KUKA KRL program: EPS_2_251349_CBMH081_A_20251001124256.src

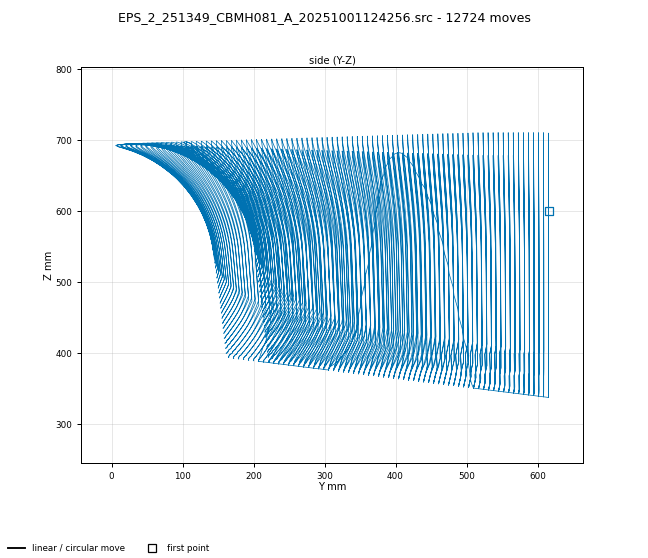
[picture p0: tool path of EPS_2_251349_CBMH081_A_20251001124256.src, 12724 of 12726 moves have a stored position in this frame; points joined in program order, loops and branches not executed]
&ACCESS RVP
&REL 4
&COMMENT QRS 19112012
&PARAM EDITMASK = *
DEF PART()
EXT BAS (BAS_COMMAND :IN,REAL :IN )
INT I
BAS (#INITMOV,0 )

;KUKA QRS Post kuka4.cps  Date:22-06-2017 !

File_ID=2858

QRS_PRE_INIT()

;Init var - Until changes are made in qrs_pre_init
Outlet_Square_prg=0
Inlet_1_Square_prg=0
Inlet_2_Square_prg=0
Inlet_3_Square_prg=0
Inlet_4_Square_prg=0
Inlet_5_Square_prg=0

Outlet_1={X 0.000, Y 517.920, Z 561.000, B 0.000, E1 0.000 }
Inlet_1={X 0.000, Y 520.260, Z 529.000, B 0.000, E1 170.000 }
Outlet_1_type=299
Inlet_1_type=299
;QRS#1=Sidecore dimensions
;QRS#2=300-12" PVC SDR 35
;QRS#3=300-12" PVC SDR 35
;QRS#4=
;QRS#5=
;QRS#6=
;QRS#7=
;QRS#8=
;QRS#9=16M PSX
;QRS#10=16M PSX
;QRS#11=
;QRS#12=
;QRS#13=
;QRS#14=
;QRS#15=
;QRS#16=1220x127x991 3,25'
;QRS#17=EPS Height
;QRS#18=710,5
;QRS#19=*
;QRS#20= UPDATED VERSION 22-06-2017
;QRS#21=*
Outlet_Square=0150
Inlet_1_Square=0150
Inlet_2_Square=0
Inlet_3_Square=0
Inlet_4_Square=0
Inlet_5_Square=0
Mill_Square=1
Outlet_Square_Prg=206
Inlet_1_Square_prg=206

QRS_INIT()

$ADVANCE=5

; T1
PTP {E1 173.61,E2 173.61}
PTP {X 0,Y 615.513,A -85,B 0,C 180,E1 173.61,E2 173.61,E3 0,E4 0,E5 0,E6 0}
QRS_SPEED_INIT()
LIN {X 0,Y 615.513,Z 600,A -85,B 0,C 180,E1 173.61,E2 173.61,E3 0,E4 0,E5 0,E6 0} C_VEL
LIN {X 0,Y 615.513,Z 347.498,A -85,B 0,C 180,E1 173.61,E2 173.61} C_VEL
LIN {X 0,Y 615.513,Z 339.324,A -85,B 0,C 180,E1 173.61,E2 173.61} C_VEL
LIN {X 0,Y 615.486,Z 337.324,A -85,B 0,C 180,E1 173.424,E2 173.424} C_VEL
LIN {X 0,Y 615.446,Z 337.318,A -85,B 0,C 180,E1 170.8,E2 170.8} C_VEL
LIN {X 0,Y 615.482,Z 337.311,A -85,B 0,C 180,E1 168.139,E2 168.139} C_VEL
LIN {X 0,Y 615.489,Z 337.325,A -85,B 0,C 180,E1 165.451,E2 165.451} C_VEL
LIN {X 0,Y 615.447,Z 337.317,A -85,B 0,C 180,E1 162.728,E2 162.728} C_VEL
LIN {X 0,Y 615.489,Z 337.312,A -85,B 0,C 180,E1 159.967,E2 159.967} C_VEL
LIN {X 0,Y 615.463,Z 337.321,A -85,B 0,C 180,E1 157.154,E2 157.154} C_VEL
LIN {X 0,Y 615.454,Z 337.32,A -85,B 0,C 180,E1 155.006,E2 155.006} C_VEL
LIN {X 0,Y 615.449,Z 337.318,A -85,B 0,C 180,E1 152.821,E2 152.821} C_VEL
LIN {X 0,Y 615.476,Z 337.311,A -85,B 0,C 180,E1 150.208,E2 150.208} C_VEL
LIN {X 0,Y 615.493,Z 337.324,A -85,B 0,C 180,E1 147.542,E2 147.542} C_VEL
LIN {X 0,Y 615.468,Z 337.322,A -85,B 0,C 180,E1 145.183,E2 145.183} C_VEL
LIN {X 0,Y 615.45,Z 337.317,A -85,B 0,C 180,E1 142.755,E2 142.755} C_VEL
LIN {X 0,Y 615.496,Z 337.311,A -85,B 0,C 180,E1 139.91,E2 139.91} C_VEL
LIN {X 0,Y 615.494,Z 337.319,A -85,B 0,C 180,E1 137.647,E2 137.647} C_VEL
LIN {X 0,Y 615.454,Z 337.319,A -85,B 0,C 180,E1 134.928,E2 134.928} C_VEL
LIN {X 0,Y 615.486,Z 337.31,A -85,B 0,C 180,E1 132.079,E2 132.079} C_VEL
LIN {X 0,Y 615.489,Z 337.317,A -85,B 0,C 180,E1 129.75,E2 129.75} C_VEL
LIN {X 0,Y 615.456,Z 337.319,A -85,B 0,C 180,E1 126.932,E2 126.932} C_VEL
LIN {X 0,Y 615.452,Z 337.316,A -85,B 0,C 180,E1 124.695,E2 124.695} C_VEL
LIN {X 0,Y 615.474,Z 337.453,A -85,B 0,C 180,E1 122.145,E2 122.145} C_VEL
LIN {X 0,Y 615.463,Z 358.452,A -85,B 0,C 180,E1 119.408,E2 119.408} C_VEL
LIN {X 0,Y 615.49,Z 368.008,A -85,B 0,C 180,E1 118.181,E2 118.181} C_VEL
LIN {X 0,Y 615.482,Z 532.764,A -85,B 0,C 180,E1 116.194,E2 116.194} C_VEL
LIN {X 0,Y 615.486,Z 547.148,A -85,B 0,C 180,E1 115.898,E2 115.898} C_VEL
LIN {X 0,Y 615.476,Z 562.128,A -85,B 0,C 180,E1 115.457,E2 115.457} C_VEL
LIN {X 0,Y 615.487,Z 576.373,A -85,B 0,C 180,E1 114.902,E2 114.902} C_VEL
LIN {X 0,Y 615.486,Z 590.475,A -85,B 0,C 180,E1 114.206,E2 114.206} C_VEL
LIN {X 0,Y 615.498,Z 602.734,A -85,B 0,C 180,E1 113.467,E2 113.467} C_VEL
LIN {X 0,Y 615.497,Z 614.806,A -85,B 0,C 180,E1 112.595,E2 112.595} C_VEL
LIN {X 0,Y 615.496,Z 626.273,A -85,B 0,C 180,E1 111.607,E2 111.607} C_VEL
LIN {X 0,Y 615.493,Z 636.516,A -85,B 0,C 180,E1 110.557,E2 110.557} C_VEL
LIN {X 0,Y 615.494,Z 646.441,A -85,B 0,C 180,E1 109.338,E2 109.338} C_VEL
LIN {X 0,Y 615.499,Z 653.657,A -85,B 0,C 180,E1 108.28,E2 108.28} C_VEL
LIN {X 0,Y 615.488,Z 661.243,A -85,B 0,C 180,E1 106.928,E2 106.928} C_VEL
LIN {X 0,Y 615.492,Z 667.287,A -85,B 0,C 180,E1 105.565,E2 105.565} C_VEL
LIN {X 0,Y 615.491,Z 670.83,A -85,B 0,C 180,E1 104.549,E2 104.549} C_VEL
LIN {X 0,Y 615.492,Z 674.376,A -85,B 0,C 180,E1 103.201,E2 103.201} C_VEL
LIN {X 0,Y 615.495,Z 676.661,A -85,B 0,C 180,E1 101.861,E2 101.861} C_VEL
LIN {X 0,Y 615.492,Z 677.759,A -85,B 0,C 180,E1 100.527,E2 100.527} C_VEL
LIN {X 0,Y 615.493,Z 677.697,A -85,B 0,C 180,E1 99.199,E2 99.199} C_VEL
LIN {X 0,Y 615.494,Z 676.457,A -85,B 0,C 180,E1 97.876,E2 97.876} C_VEL
LIN {X 0,Y 615.49,Z 674.047,A -85,B 0,C 180,E1 96.557,E2 96.557} C_VEL
LIN {X 0,Y 615.491,Z 670.446,A -85,B 0,C 180,E1 95.241,E2 95.241} C_VEL
LIN {X 0,Y 615.496,Z 665.591,A -85,B 0,C 180,E1 93.928,E2 93.928} C_VEL
LIN {X 0,Y 615.493,Z 659.363,A -85,B 0,C 180,E1 92.618,E2 92.618} C_VEL
LIN {X 0,Y 615.49,Z 651.592,A -85,B 0,C 180,E1 91.309,E2 91.309} C_VEL
LIN {X 0,Y 615.499,Z 643.35,A -85,B 0,C 180,E1 90.164,E2 90.164} C_VEL
LIN {X 0,Y 615.496,Z 633.468,A -85,B 0,C 180,E1 89.019,E2 89.019} C_VEL
LIN {X 0,Y 615.5,Z 623.429,A -85,B 0,C 180,E1 88.037,E2 88.037} C_VEL
LIN {X 0,Y 615.498,Z 611.464,A -85,B 0,C 180,E1 87.055,E2 87.055} C_VEL
LIN {X 0,Y 615.5,Z 599.577,A -85,B 0,C 180,E1 86.235,E2 86.235} C_VEL
LIN {X 0,Y 615.475,Z 586.657,A -85,B 0,C 180,E1 85.497,E2 85.497} C_VEL
LIN {X 0,Y 615.487,Z 572.479,A -85,B 0,C 180,E1 84.841,E2 84.841} C_VEL
LIN {X 0,Y 615.484,Z 557.682,A -85,B 0,C 180,E1 84.307,E2 84.307} C_VEL
LIN {X 0,Y 615.49,Z 543.934,A -85,B 0,C 180,E1 83.938,E2 83.938} C_VEL
LIN {X 0,Y 615.479,Z 529.603,A -85,B 0,C 180,E1 83.672,E2 83.672} C_VEL
LIN {X 0,Y 615.486,Z 367.825,A -85,B 0,C 180,E1 81.711,E2 81.711} C_VEL
LIN {X 0,Y 615.46,Z 346.644,A -85,B 0,C 180,E1 78.968,E2 78.968} C_VEL
LIN {X 0,Y 615.466,Z 337.313,A -85,B 0,C 180,E1 77.721,E2 77.721} C_VEL
LIN {X 0,Y 615.45,Z 337.315,A -85,B 0,C 180,E1 75.45,E2 75.45} C_VEL
LIN {X 0,Y 615.449,Z 337.316,A -85,B 0,C 180,E1 73.412,E2 73.412} C_VEL
LIN {X 0,Y 615.447,Z 337.316,A -85,B 0,C 180,E1 71.353,E2 71.353} C_VEL
LIN {X 0,Y 615.445,Z 337.317,A -85,B 0,C 180,E1 69.268,E2 69.268} C_VEL
LIN {X 0,Y 615.446,Z 337.318,A -85,B 0,C 180,E1 67.154,E2 67.154} C_VEL
LIN {X 0,Y 615.499,Z 337.324,A -85,B 0,C 180,E1 64.43,E2 64.43} C_VEL
LIN {X 0,Y 615.455,Z 337.314,A -85,B 0,C 180,E1 61.556,E2 61.556} C_VEL
LIN {X 0,Y 615.445,Z 337.32,A -85,B 0,C 180,E1 59.078,E2 59.078} C_VEL
LIN {X 0,Y 615.495,Z 337.326,A -85,B 0,C 180,E1 56.466,E2 56.466} C_VEL
LIN {X 0,Y 615.456,Z 337.314,A -85,B 0,C 180,E1 53.573,E2 53.573} C_VEL
LIN {X 0,Y 615.45,Z 337.321,A -85,B 0,C 180,E1 50.943,E2 50.943} C_VEL
LIN {X 0,Y 615.486,Z 337.325,A -85,B 0,C 180,E1 48.526,E2 48.526} C_VEL
LIN {X 0,Y 615.481,Z 337.312,A -85,B 0,C 180,E1 45.85,E2 45.85} C_VEL
LIN {X 0,Y 615.444,Z 337.317,A -85,B 0,C 180,E1 43.249,E2 43.249} C_VEL
LIN {X 0,Y 615.479,Z 337.324,A -85,B 0,C 180,E1 40.608,E2 40.608} C_VEL
LIN {X 0,Y 615.483,Z 337.315,A -85,B 0,C 180,E1 38.011,E2 38.011} C_VEL
LIN {X 0,Y 615.458,Z 337.314,A -85,B 0,C 180,E1 35.618,E2 35.618} C_VEL
LIN {X 0,Y 615.441,Z 337.318,A -85,B 0,C 180,E1 33.24,E2 33.24} C_VEL
LIN {X 0,Y 615.451,Z 337.321,A -85,B 0,C 180,E1 30.922,E2 30.922} C_VEL
LIN {X 0,Y 615.497,Z 337.325,A -85,B 0,C 180,E1 28.451,E2 28.451} C_VEL
LIN {X 0,Y 615.454,Z 337.315,A -85,B 0,C 180,E1 25.562,E2 25.562} C_VEL
LIN {X 0,Y 615.453,Z 337.315,A -85,B 0,C 180,E1 23.558,E2 23.558} C_VEL
LIN {X 0,Y 615.447,Z 337.316,A -85,B 0,C 180,E1 21.434,E2 21.434} C_VEL
LIN {X 0,Y 615.444,Z 337.317,A -85,B 0,C 180,E1 19.34,E2 19.34} C_VEL
LIN {X 0,Y 615.442,Z 337.317,A -85,B 0,C 180,E1 17.272,E2 17.272} C_VEL
LIN {X 0,Y 615.482,Z 337.324,A -85,B 0,C 180,E1 14.55,E2 14.55} C_VEL
LIN {X 0,Y 615.482,Z 337.312,A -85,B 0,C 180,E1 11.861,E2 11.861} C_VEL
LIN {X 0,Y 615.441,Z 337.318,A -85,B 0,C 180,E1 9.2,E2 9.2} C_VEL
LIN {X 0,Y 615.48,Z 337.324,A -85,B 0,C 180,E1 6.557,E2 6.557} C_VEL
LIN {X 0,Y 615.483,Z 337.314,A -85,B 0,C 180,E1 3.929,E2 3.929} C_VEL
LIN {X 0,Y 615.442,Z 337.317,A -85,B 0,C 180,E1 1.309,E2 1.309} C_VEL
LIN {X 0,Y 615.465,Z 337.323,A -85,B 0,C 180,E1 -1.308,E2 -1.308} C_VEL
LIN {X 0,Y 615.491,Z 337.316,A -85,B 0,C 180,E1 -3.928,E2 -3.928} C_VEL
LIN {X 0,Y 615.446,Z 337.316,A -85,B 0,C 180,E1 -6.557,E2 -6.557} C_VEL
LIN {X 0,Y 615.447,Z 337.316,A -85,B 0,C 180,E1 -8.537,E2 -8.537} C_VEL
LIN {X 0,Y 615.44,Z 337.319,A -85,B 0,C 180,E1 -10.864,E2 -10.864} C_VEL
LIN {X 0,Y 615.454,Z 337.322,A -85,B 0,C 180,E1 -13.202,E2 -13.202} C_VEL
LIN {X 0,Y 615.494,Z 337.316,A -85,B 0,C 180,E1 -15.905,E2 -15.905} C_VEL
LIN {X 0,Y 615.442,Z 337.317,A -85,B 0,C 180,E1 -18.647,E2 -18.647} C_VEL
LIN {X 0,Y 615.44,Z 337.318,A -85,B 0,C 180,E1 -20.732,E2 -20.732} C_VEL
LIN {X 0,Y 615.439,Z 337.319,A -85,B 0,C 180,E1 -22.846,E2 -22.846} C_VEL
LIN {X 0,Y 615.442,Z 337.32,A -85,B 0,C 180,E1 -24.994,E2 -24.994} C_VEL
LIN {X 0,Y 615.49,Z 337.317,A -85,B 0,C 180,E1 -27.915,E2 -27.915} C_VEL
LIN {X 0,Y 615.479,Z 337.313,A -85,B 0,C 180,E1 -30.16,E2 -30.16} C_VEL
LIN {X 0,Y 615.45,Z 337.316,A -85,B 0,C 180,E1 -32.459,E2 -32.459} C_VEL
LIN {X 0,Y 615.437,Z 337.319,A -85,B 0,C 180,E1 -34.818,E2 -34.818} C_VEL
LIN {X 0,Y 615.452,Z 337.323,A -85,B 0,C 180,E1 -37.245,E2 -37.245} C_VEL
LIN {X 0,Y 615.488,Z 337.313,A -85,B 0,C 180,E1 -40.089,E2 -40.089} C_VEL
LIN {X 0,Y 615.458,Z 337.315,A -85,B 0,C 180,E1 -42.355,E2 -42.355} C_VEL
LIN {X 0,Y 615.439,Z 337.32,A -85,B 0,C 180,E1 -44.927,E2 -44.927} C_VEL
LIN {X 0,Y 615.499,Z 337.325,A -85,B 0,C 180,E1 -47.648,E2 -47.648} C_VEL
LIN {X 0,Y 615.467,Z 337.315,A -85,B 0,C 180,E1 -50.248,E2 -50.248} C_VEL
LIN {X 0,Y 615.437,Z 337.318,A -85,B 0,C 180,E1 -52.754,E2 -52.754} C_VEL
LIN {X 0,Y 615.458,Z 337.322,A -85,B 0,C 180,E1 -55.303,E2 -55.303} C_VEL
LIN {X 0,Y 615.461,Z 337.315,A -85,B 0,C 180,E1 -58.313,E2 -58.313} C_VEL
LIN {X 0,Y 615.442,Z 337.317,A -85,B 0,C 180,E1 -60.591,E2 -60.591} C_VEL
LIN {X 0,Y 615.438,Z 337.32,A -85,B 0,C 180,E1 -62.964,E2 -62.964} C_VEL
LIN {X 0,Y 615.436,Z 337.373,A -85,B 0,C 180,E1 -64.846,E2 -64.846} C_VEL
LIN {X 0,Y 615.479,Z 359.775,A -85,B 0,C 180,E1 -67.404,E2 -67.404} C_VEL
LIN {X 0,Y 615.49,Z 384.221,A -85,B 0,C 180,E1 -70.141,E2 -70.141} C_VEL
LIN {X 0,Y 615.488,Z 399.033,A -85,B 0,C 180,E1 -71.762,E2 -71.762} C_VEL
LIN {X 0,Y 615.484,Z 565.218,A -85,B 0,C 180,E1 -73.769,E2 -73.769} C_VEL
LIN {X 0,Y 615.49,Z 580.71,A -85,B 0,C 180,E1 -74.095,E2 -74.095} C_VEL
LIN {X 0,Y 615.48,Z 596.048,A -85,B 0,C 180,E1 -74.562,E2 -74.562} C_VEL
LIN {X 0,Y 615.484,Z 609.752,A -85,B 0,C 180,E1 -75.113,E2 -75.113} C_VEL
LIN {X 0,Y 615.493,Z 624.045,A -85,B 0,C 180,E1 -75.833,E2 -75.833} C_VEL
LIN {X 0,Y 615.497,Z 636.897,A -85,B 0,C 180,E1 -76.631,E2 -76.631} C_VEL
LIN {X 0,Y 615.495,Z 649.254,A -85,B 0,C 180,E1 -77.554,E2 -77.554} C_VEL
LIN {X 0,Y 615.495,Z 659.606,A -85,B 0,C 180,E1 -78.473,E2 -78.473} C_VEL
LIN {X 0,Y 615.494,Z 669.183,A -85,B 0,C 180,E1 -79.473,E2 -79.473} C_VEL
LIN {X 0,Y 615.493,Z 678.577,A -85,B 0,C 180,E1 -80.636,E2 -80.636} C_VEL
LIN {X 0,Y 615.497,Z 686.38,A -85,B 0,C 180,E1 -81.794,E2 -81.794} C_VEL
LIN {X 0,Y 615.494,Z 693.609,A -85,B 0,C 180,E1 -83.102,E2 -83.102} C_VEL
LIN {X 0,Y 615.499,Z 699.436,A -85,B 0,C 180,E1 -84.43,E2 -84.43} C_VEL
LIN {X 0,Y 615.491,Z 702.86,A -85,B 0,C 180,E1 -85.415,E2 -85.415} C_VEL
LIN {X 0,Y 615.493,Z 706.318,A -85,B 0,C 180,E1 -86.727,E2 -86.727} C_VEL
LIN {X 0,Y 615.499,Z 708.593,A -85,B 0,C 180,E1 -88.037,E2 -88.037} C_VEL
LIN {X 0,Y 615.491,Z 709.741,A -85,B 0,C 180,E1 -89.346,E2 -89.346} C_VEL
LIN {X 0,Y 615.491,Z 709.741,A -85,B 0,C 180,E1 -90.654,E2 -90.654} C_VEL
LIN {X 0,Y 615.499,Z 708.593,A -85,B 0,C 180,E1 -91.963,E2 -91.963} C_VEL
LIN {X 0,Y 615.493,Z 706.318,A -85,B 0,C 180,E1 -93.273,E2 -93.273} C_VEL
LIN {X 0,Y 615.491,Z 702.86,A -85,B 0,C 180,E1 -94.584,E2 -94.584} C_VEL
LIN {X 0,Y 615.497,Z 698.142,A -85,B 0,C 180,E1 -95.898,E2 -95.898} C_VEL
LIN {X 0,Y 615.492,Z 692.03,A -85,B 0,C 180,E1 -97.216,E2 -97.216} C_VEL
LIN {X 0,Y 615.49,Z 684.333,A -85,B 0,C 180,E1 -98.537,E2 -98.537} C_VEL
LIN {X 0,Y 615.495,Z 676.114,A -85,B 0,C 180,E1 -99.696,E2 -99.696} C_VEL
LIN {X 0,Y 615.496,Z 665.898,A -85,B 0,C 180,E1 -100.892,E2 -100.892} C_VEL
LIN {X 0,Y 615.496,Z 656.067,A -85,B 0,C 180,E1 -101.861,E2 -101.861} C_VEL
LIN {X 0,Y 615.497,Z 643.947,A -85,B 0,C 180,E1 -102.865,E2 -102.865} C_VEL
LIN {X 0,Y 615.498,Z 631.797,A -85,B 0,C 180,E1 -103.706,E2 -103.706} C_VEL
LIN {X 0,Y 615.477,Z 618.379,A -85,B 0,C 180,E1 -104.473,E2 -104.473} C_VEL
LIN {X 0,Y 615.495,Z 603.847,A -85,B 0,C 180,E1 -105.141,E2 -105.141} C_VEL
LIN {X 0,Y 615.48,Z 589.615,A -85,B 0,C 180,E1 -105.65,E2 -105.65} C_VEL
LIN {X 0,Y 615.499,Z 575.154,A -85,B 0,C 180,E1 -106.035,E2 -106.035} C_VEL
LIN {X 0,Y 615.48,Z 560.677,A -85,B 0,C 180,E1 -106.296,E2 -106.296} C_VEL
LIN {X 0,Y 615.491,Z 398.712,A -85,B 0,C 180,E1 -108.258,E2 -108.258} C_VEL
LIN {X 0,Y 615.487,Z 373.248,A -85,B 0,C 180,E1 -111.081,E2 -111.081} C_VEL
LIN {X 0,Y 615.487,Z 349.309,A -85,B 0,C 180,E1 -113.783,E2 -113.783} C_VEL
LIN {X 0,Y 615.436,Z 337.319,A -85,B 0,C 180,E1 -115.171,E2 -115.171} C_VEL
LIN {X 0,Y 615.436,Z 337.319,A -85,B 0,C 180,E1 -117.18,E2 -117.18} C_VEL
LIN {X 0,Y 615.472,Z 337.314,A -85,B 0,C 180,E1 -119.792,E2 -119.792} C_VEL
LIN {X 0,Y 615.486,Z 337.324,A -85,B 0,C 180,E1 -122.458,E2 -122.458} C_VEL
LIN {X 0,Y 615.45,Z 337.322,A -85,B 0,C 180,E1 -124.818,E2 -124.818} C_VEL
LIN {X 0,Y 615.438,Z 337.318,A -85,B 0,C 180,E1 -127.246,E2 -127.246} C_VEL
LIN {X 0,Y 615.496,Z 337.316,A -85,B 0,C 180,E1 -130.09,E2 -130.09} C_VEL
LIN {X 0,Y 615.498,Z 337.325,A -85,B 0,C 180,E1 -132.352,E2 -132.352} C_VEL
LIN {X 0,Y 615.44,Z 337.319,A -85,B 0,C 180,E1 -135.073,E2 -135.073} C_VEL
LIN {X 0,Y 615.485,Z 337.313,A -85,B 0,C 180,E1 -137.92,E2 -137.92} C_VEL
LIN {X 0,Y 615.496,Z 337.321,A -85,B 0,C 180,E1 -140.251,E2 -140.251} C_VEL
LIN {X 0,Y 615.441,Z 337.319,A -85,B 0,C 180,E1 -143.069,E2 -143.069} C_VEL
LIN {X 0,Y 615.441,Z 337.317,A -85,B 0,C 180,E1 -145.306,E2 -145.306} C_VEL
LIN {X 0,Y 615.459,Z 337.315,A -85,B 0,C 180,E1 -147.674,E2 -147.674} C_VEL
LIN {X 0,Y 615.476,Z 337.323,A -85,B 0,C 180,E1 -150.593,E2 -150.593} C_VEL
LIN {X 0,Y 615.447,Z 337.32,A -85,B 0,C 180,E1 -152.963,E2 -152.963} C_VEL
LIN {X 0,Y 615.445,Z 337.32,A -85,B 0,C 180,E1 -155.007,E2 -155.007} C_VEL
LIN {X 0,Y 615.461,Z 337.314,A -85,B 0,C 180,E1 -157.661,E2 -157.661} C_VEL
LIN {X 0,Y 615.471,Z 337.323,A -85,B 0,C 180,E1 -160.662,E2 -160.662} C_VEL
LIN {X 0,Y 615.465,Z 337.322,A -85,B 0,C 180,E1 -162.729,E2 -162.729} C_VEL
LIN {X 0,Y 615.461,Z 337.322,A -85,B 0,C 180,E1 -164.774,E2 -164.774} C_VEL
LIN {X 0,Y 615.459,Z 337.322,A -85,B 0,C 180,E1 -166.798,E2 -166.798} C_VEL
LIN {X 0,Y 615.444,Z 337.319,A -85,B 0,C 180,E1 -169.134,E2 -169.134} C_VEL
LIN {X 0,Y 615.449,Z 337.315,A -85,B 0,C 180,E1 -171.463,E2 -171.463} C_VEL
LIN {X 0,Y 615.496,Z 337.314,A -85,B 0,C 180,E1 -174.102,E2 -174.102} C_VEL
LIN {X 0,Y 615.468,Z 337.322,A -85,B 0,C 180,E1 -176.727,E2 -176.727} C_VEL
LIN {X 0,Y 615.472,Z 337.323,A -85,B 0,C 180,E1 -178.692,E2 -178.692} C_VEL
LIN {X 0,Y 615.445,Z 337.317,A -85,B 0,C 180,E1 -181.309,E2 -181.309} C_VEL
LIN {X 0,Y 615.483,Z 337.312,A -85,B 0,C 180,E1 -183.929,E2 -183.929} C_VEL
LIN {X 0,Y 615.486,Z 337.324,A -85,B 0,C 180,E1 -186.576,E2 -186.576} C_VEL
LIN {X 0,Y 614.781,Z 337.464,A -85,B 0,C 180,E1 -187.122,E2 -187.122} C_VEL
LIN {X 0,Y 611.924,Z 337.883,A -85,B 0,C 180,E1 -188.007,E2 -188.007} C_VEL
LIN {X 0,Y 609.538,Z 338.19,A -85,B 0,C 180,E1 -188.72,E2 -188.72} C_VEL
LIN {X 0,Y 608.517,Z 338.305,A -85,B 0,C 180,E1 -189.27,E2 -189.27} C_VEL
LIN {X 0,Y 608.435,Z 338.314,A -85,B 0,C 180,E1 -189.456,E2 -189.456} C_VEL
LIN {X 0,Y 608.459,Z 338.314,A -85,B 0,C 180,E1 -192,E2 -192} C_VEL
LIN {X 0,Y 608.468,Z 338.317,A -85,B 0,C 180,E1 -194.721,E2 -194.721} C_VEL
LIN {X 0,Y 608.43,Z 338.315,A -85,B 0,C 180,E1 -197.478,E2 -197.478} C_VEL
LIN {X 0,Y 608.431,Z 338.314,A -85,B 0,C 180,E1 -199.572,E2 -199.572} C_VEL
LIN {X 0,Y 608.481,Z 338.318,A -85,B 0,C 180,E1 -202.405,E2 -202.405} C_VEL
LIN {X 0,Y 608.446,Z 338.322,A -85,B 0,C 180,E1 -204.572,E2 -204.572} C_VEL
LIN {X 0,Y 608.43,Z 338.316,A -85,B 0,C 180,E1 -207.198,E2 -207.198} C_VEL
LIN {X 0,Y 608.461,Z 338.312,A -85,B 0,C 180,E1 -209.78,E2 -209.78} C_VEL
LIN {X 0,Y 608.466,Z 338.322,A -85,B 0,C 180,E1 -212.523,E2 -212.523} C_VEL
LIN {X 0,Y 608.424,Z 338.316,A -85,B 0,C 180,E1 -215.279,E2 -215.279} C_VEL
LIN {X 0,Y 608.467,Z 338.316,A -85,B 0,C 180,E1 -218.24,E2 -218.24} C_VEL
LIN {X 0,Y 608.42,Z 338.317,A -85,B 0,C 180,E1 -221.18,E2 -221.18} C_VEL
LIN {X 0,Y 608.466,Z 338.312,A -85,B 0,C 180,E1 -223.87,E2 -223.87} C_VEL
LIN {X 0,Y 608.466,Z 338.319,A -85,B 0,C 180,E1 -226.692,E2 -226.692} C_VEL
LIN {X 0,Y 608.44,Z 338.32,A -85,B 0,C 180,E1 -228.822,E2 -228.822} C_VEL
LIN {X 0,Y 608.46,Z 338.312,A -85,B 0,C 180,E1 -231.761,E2 -231.761} C_VEL
LIN {X 0,Y 608.436,Z 338.322,A -85,B 0,C 180,E1 -234.722,E2 -234.722} C_VEL
LIN {X 0,Y 608.444,Z 338.316,A -85,B 0,C 180,E1 -237.12,E2 -237.12} C_VEL
LIN {X 0,Y 608.481,Z 338.475,A -85,B 0,C 180,E1 -237.722,E2 -237.722} C_VEL
LIN {X 0,Y 608.527,Z 357.408,A -85,B 0,C 180,E1 -240.224,E2 -240.224} C_VEL
LIN {X 0,Y 608.538,Z 367.98,A -85,B 0,C 180,E1 -241.603,E2 -241.603} C_VEL
LIN {X 0,Y 608.768,Z 378.048,A -85,B 0,C 180,E1 -241.732,E2 -241.732} C_VEL
LIN {X 0,Y 608.676,Z 533.346,A -85,B 0,C 180,E1 -243.629,E2 -243.629} C_VEL
LIN {X 0,Y 608.665,Z 549.358,A -85,B 0,C 180,E1 -243.975,E2 -243.975} C_VEL
LIN {X 0,Y 608.618,Z 563.717,A -85,B 0,C 180,E1 -244.416,E2 -244.416} C_VEL
LIN {X 0,Y 608.592,Z 577.624,A -85,B 0,C 180,E1 -244.979,E2 -244.979} C_VEL
LIN {X 0,Y 608.557,Z 591.482,A -85,B 0,C 180,E1 -245.682,E2 -245.682} C_VEL
LIN {X 0,Y 608.545,Z 604.931,A -85,B 0,C 180,E1 -246.52,E2 -246.52} C_VEL
LIN {X 0,Y 608.528,Z 617.115,A -85,B 0,C 180,E1 -247.436,E2 -247.436} C_VEL
LIN {X 0,Y 608.486,Z 628.833,A -85,B 0,C 180,E1 -248.487,E2 -248.487} C_VEL
LIN {X 0,Y 608.475,Z 639.142,A -85,B 0,C 180,E1 -249.594,E2 -249.594} C_VEL
LIN {X 0,Y 608.467,Z 648.398,A -85,B 0,C 180,E1 -250.781,E2 -250.781} C_VEL
LIN {X 0,Y 608.464,Z 656.297,A -85,B 0,C 180,E1 -252.003,E2 -252.003} C_VEL
LIN {X 0,Y 608.453,Z 662.751,A -85,B 0,C 180,E1 -253.216,E2 -253.216} C_VEL
LIN {X 0,Y 608.423,Z 668.603,A -85,B 0,C 180,E1 -254.593,E2 -254.593} C_VEL
LIN {X 0,Y 608.446,Z 673.082,A -85,B 0,C 180,E1 -255.994,E2 -255.994} C_VEL
LIN {X 0,Y 608.417,Z 676.06,A -85,B 0,C 180,E1 -257.322,E2 -257.322} C_VEL
LIN {X 0,Y 608.427,Z 677.88,A -85,B 0,C 180,E1 -258.675,E2 -258.675} C_VEL
LIN {X 0,Y 608.43,Z 678.499,A -85,B 0,C 180,E1 -260.022,E2 -260.022} C_VEL
LIN {X 0,Y 608.414,Z 677.916,A -85,B 0,C 180,E1 -261.363,E2 -261.363} C_VEL
LIN {X 0,Y 608.418,Z 676.173,A -85,B 0,C 180,E1 -262.7,E2 -262.7} C_VEL
LIN {X 0,Y 608.433,Z 673.251,A -85,B 0,C 180,E1 -264.033,E2 -264.033} C_VEL
LIN {X 0,Y 608.428,Z 669.105,A -85,B 0,C 180,E1 -265.362,E2 -265.362} C_VEL
LIN {X 0,Y 608.431,Z 663.65,A -85,B 0,C 180,E1 -266.689,E2 -266.689} C_VEL
LIN {X 0,Y 608.467,Z 656.739,A -85,B 0,C 180,E1 -268.014,E2 -268.014} C_VEL
LIN {X 0,Y 608.467,Z 648.185,A -85,B 0,C 180,E1 -269.338,E2 -269.338} C_VEL
LIN {X 0,Y 608.468,Z 639.143,A -85,B 0,C 180,E1 -270.496,E2 -270.496} C_VEL
LIN {X 0,Y 608.489,Z 628.289,A -85,B 0,C 180,E1 -271.655,E2 -271.655} C_VEL
LIN {X 0,Y 608.526,Z 617.195,A -85,B 0,C 180,E1 -272.648,E2 -272.648} C_VEL
LIN {X 0,Y 608.539,Z 605.104,A -85,B 0,C 180,E1 -273.559,E2 -273.559} C_VEL
LIN {X 0,Y 608.571,Z 591.843,A -85,B 0,C 180,E1 -274.388,E2 -274.388} C_VEL
LIN {X 0,Y 608.592,Z 578.944,A -85,B 0,C 180,E1 -275.052,E2 -275.052} C_VEL
LIN {X 0,Y 608.631,Z 564.807,A -85,B 0,C 180,E1 -275.633,E2 -275.633} C_VEL
LIN {X 0,Y 608.645,Z 549.57,A -85,B 0,C 180,E1 -276.11,E2 -276.11} C_VEL
LIN {X 0,Y 608.668,Z 534.404,A -85,B 0,C 180,E1 -276.441,E2 -276.441} C_VEL
LIN {X 0,Y 608.671,Z 500.168,A -85,B 0,C 180,E1 -276.88,E2 -276.88} C_VEL
LIN {X 0,Y 608.635,Z 368.605,A -85,B 0,C 180,E1 -278.477,E2 -278.477} C_VEL
LIN {X 0,Y 608.524,Z 367.812,A -85,B 0,C 180,E1 -278.51,E2 -278.51} C_VEL
LIN {X 0,Y 608.551,Z 347.627,A -85,B 0,C 180,E1 -281.152,E2 -281.152} C_VEL
LIN {X 0,Y 608.436,Z 338.316,A -85,B 0,C 180,E1 -282.402,E2 -282.402} C_VEL
LIN {X 0,Y 608.418,Z 338.317,A -85,B 0,C 180,E1 -284.722,E2 -284.722} C_VEL
LIN {X 0,Y 608.445,Z 338.323,A -85,B 0,C 180,E1 -287.477,E2 -287.477} C_VEL
LIN {X 0,Y 608.447,Z 338.313,A -85,B 0,C 180,E1 -290.275,E2 -290.275} C_VEL
LIN {X 0,Y 608.435,Z 338.314,A -85,B 0,C 180,E1 -292.469,E2 -292.469} C_VEL
LIN {X 0,Y 608.431,Z 338.315,A -85,B 0,C 180,E1 -294.572,E2 -294.572} C_VEL
LIN {X 0,Y 608.458,Z 338.316,A -85,B 0,C 180,E1 -297.202,E2 -297.202} C_VEL
LIN {X 0,Y 608.471,Z 338.313,A -85,B 0,C 180,E1 -299.971,E2 -299.971} C_VEL
LIN {X 0,Y 608.437,Z 338.315,A -85,B 0,C 180,E1 -302.881,E2 -302.881} C_VEL
LIN {X 0,Y 608.435,Z 338.32,A -85,B 0,C 180,E1 -305.278,E2 -305.278} C_VEL
LIN {X 0,Y 608.46,Z 338.312,A -85,B 0,C 180,E1 -308.239,E2 -308.239} C_VEL
LIN {X 0,Y 608.43,Z 338.319,A -85,B 0,C 180,E1 -311.179,E2 -311.179} C_VEL
LIN {X 0,Y 608.468,Z 338.315,A -85,B 0,C 180,E1 -313.87,E2 -313.87} C_VEL
LIN {X 0,Y 608.438,Z 338.314,A -85,B 0,C 180,E1 -316.695,E2 -316.695} C_VEL
LIN {X 0,Y 608.415,Z 338.317,A -85,B 0,C 180,E1 -318.82,E2 -318.82} C_VEL
LIN {X 0,Y 608.464,Z 338.318,A -85,B 0,C 180,E1 -321.76,E2 -321.76} C_VEL
LIN {X 0,Y 608.419,Z 338.316,A -85,B 0,C 180,E1 -324.72,E2 -324.72} C_VEL
LIN {X 0,Y 608.465,Z 338.32,A -85,B 0,C 180,E1 -327.478,E2 -327.478} C_VEL
LIN {X 0,Y 608.46,Z 338.312,A -85,B 0,C 180,E1 -330.22,E2 -330.22} C_VEL
LIN {X 0,Y 608.423,Z 338.316,A -85,B 0,C 180,E1 -332.803,E2 -332.803} C_VEL
LIN {X 0,Y 608.443,Z 338.321,A -85,B 0,C 180,E1 -335.428,E2 -335.428} C_VEL
LIN {X 0,Y 608.451,Z 338.313,A -85,B 0,C 180,E1 -338.307,E2 -338.307} C_VEL
LIN {X 0,Y 608.443,Z 338.317,A -85,B 0,C 180,E1 -341.13,E2 -341.13} C_VEL
LIN {X 0,Y 608.461,Z 338.316,A -85,B 0,C 180,E1 -343.906,E2 -343.906} C_VEL
LIN {X 0,Y 608.432,Z 338.315,A -85,B 0,C 180,E1 -346.643,E2 -346.643} C_VEL
LIN {X 0,Y 608.452,Z 338.318,A -85,B 0,C 180,E1 -349.35,E2 -349.35} C_VEL
LIN {X 0,Y 608.474,Z 338.313,A -85,B 0,C 180,E1 -352.033,E2 -352.033} C_VEL
LIN {X 0,Y 608.427,Z 338.315,A -85,B 0,C 180,E1 -354.697,E2 -354.697} C_VEL
LIN {X 0,Y 608.464,Z 338.317,A -85,B 0,C 180,E1 -357.352,E2 -357.352} C_VEL
LIN {X 0,Y 608.477,Z 338.313,A -85,B 0,C 180,E1 -360,E2 -360} C_VEL
LIN {X 0,Y 608.439,Z 338.313,A -85,B 0,C 180,E1 -362.648,E2 -362.648} C_VEL
LIN {X 0,Y 608.443,Z 338.319,A -85,B 0,C 180,E1 -365.302,E2 -365.302} C_VEL
LIN {X 0,Y 608.48,Z 338.313,A -85,B 0,C 180,E1 -367.967,E2 -367.967} C_VEL
LIN {X 0,Y 608.439,Z 338.315,A -85,B 0,C 180,E1 -370.939,E2 -370.939} C_VEL
LIN {X 0,Y 608.443,Z 338.319,A -85,B 0,C 180,E1 -373.357,E2 -373.357} C_VEL
LIN {X 0,Y 608.454,Z 338.315,A -85,B 0,C 180,E1 -376.094,E2 -376.094} C_VEL
LIN {X 0,Y 608.435,Z 338.315,A -85,B 0,C 180,E1 -378.87,E2 -378.87} C_VEL
LIN {X 0,Y 608.461,Z 338.321,A -85,B 0,C 180,E1 -381.692,E2 -381.692} C_VEL
LIN {X 0,Y 608.428,Z 338.315,A -85,B 0,C 180,E1 -384.572,E2 -384.572} C_VEL
LIN {X 0,Y 608.45,Z 338.316,A -85,B 0,C 180,E1 -387.202,E2 -387.202} C_VEL
LIN {X 0,Y 608.471,Z 338.315,A -85,B 0,C 180,E1 -389.972,E2 -389.972} C_VEL
LIN {X 0,Y 608.43,Z 338.315,A -85,B 0,C 180,E1 -392.881,E2 -392.881} C_VEL
LIN {X 0,Y 608.432,Z 338.319,A -85,B 0,C 180,E1 -395.278,E2 -395.278} C_VEL
LIN {X 0,Y 608.458,Z 338.313,A -85,B 0,C 180,E1 -398.239,E2 -398.239} C_VEL
LIN {X 0,Y 608.42,Z 338.319,A -85,B 0,C 180,E1 -401.179,E2 -401.179} C_VEL
LIN {X 0,Y 608.466,Z 338.317,A -85,B 0,C 180,E1 -403.87,E2 -403.87} C_VEL
LIN {X 0,Y 608.432,Z 338.315,A -85,B 0,C 180,E1 -406.695,E2 -406.695} C_VEL
LIN {X 0,Y 608.409,Z 338.318,A -85,B 0,C 180,E1 -408.819,E2 -408.819} C_VEL
LIN {X 0,Y 608.463,Z 338.32,A -85,B 0,C 180,E1 -411.76,E2 -411.76} C_VEL
LIN {X 0,Y 608.414,Z 338.317,A -85,B 0,C 180,E1 -414.72,E2 -414.72} C_VEL
LIN {X 0,Y 608.459,Z 338.319,A -85,B 0,C 180,E1 -417.478,E2 -417.478} C_VEL
LIN {X 0,Y 608.458,Z 338.314,A -85,B 0,C 180,E1 -420.22,E2 -420.22} C_VEL
LIN {X 0,Y 608.418,Z 338.317,A -85,B 0,C 180,E1 -422.804,E2 -422.804} C_VEL
LIN {X 0,Y 608.433,Z 338.45,A -85,B 0,C 180,E1 -424.662,E2 -424.662} C_VEL
LIN {X 0,Y 608.66,Z 349.305,A -85,B 0,C 180,E1 -425.933,E2 -425.933} C_VEL
LIN {X 0,Y 608.619,Z 373.247,A -85,B 0,C 180,E1 -428.67,E2 -428.67} C_VEL
LIN {X 0,Y 608.551,Z 398.721,A -85,B 0,C 180,E1 -431.526,E2 -431.526} C_VEL
LIN {X 0,Y 608.752,Z 404.044,A -85,B 0,C 180,E1 -431.614,E2 -431.614} C_VEL
LIN {X 0,Y 608.678,Z 565.217,A -85,B 0,C 180,E1 -433.582,E2 -433.582} C_VEL
LIN {X 0,Y 608.651,Z 580.709,A -85,B 0,C 180,E1 -433.911,E2 -433.911} C_VEL
LIN {X 0,Y 608.618,Z 596.047,A -85,B 0,C 180,E1 -434.383,E2 -434.383} C_VEL
LIN {X 0,Y 608.605,Z 609.754,A -85,B 0,C 180,E1 -434.94,E2 -434.94} C_VEL
LIN {X 0,Y 608.572,Z 623.235,A -85,B 0,C 180,E1 -435.624,E2 -435.624} C_VEL
LIN {X 0,Y 608.554,Z 635.663,A -85,B 0,C 180,E1 -436.39,E2 -436.39} C_VEL
LIN {X 0,Y 608.528,Z 648.282,A -85,B 0,C 180,E1 -437.324,E2 -437.324} C_VEL
LIN {X 0,Y 608.496,Z 659.747,A -85,B 0,C 180,E1 -438.339,E2 -438.339} C_VEL
LIN {X 0,Y 608.475,Z 669.387,A -85,B 0,C 180,E1 -439.35,E2 -439.35} C_VEL
LIN {X 0,Y 608.476,Z 678.853,A -85,B 0,C 180,E1 -440.527,E2 -440.527} C_VEL
LIN {X 0,Y 608.457,Z 686.729,A -85,B 0,C 180,E1 -441.698,E2 -441.698} C_VEL
LIN {X 0,Y 608.439,Z 694.087,A -85,B 0,C 180,E1 -443.034,E2 -443.034} C_VEL
LIN {X 0,Y 608.45,Z 699.923,A -85,B 0,C 180,E1 -444.366,E2 -444.366} C_VEL
LIN {X 0,Y 608.427,Z 703.383,A -85,B 0,C 180,E1 -445.362,E2 -445.362} C_VEL
LIN {X 0,Y 608.421,Z 706.885,A -85,B 0,C 180,E1 -446.689,E2 -446.689} C_VEL
LIN {X 0,Y 608.444,Z 709.191,A -85,B 0,C 180,E1 -448.014,E2 -448.014} C_VEL
LIN {X 0,Y 608.434,Z 710.351,A -85,B 0,C 180,E1 -449.338,E2 -449.338} C_VEL
LIN {X 0,Y 608.434,Z 710.351,A -85,B 0,C 180,E1 -450.662,E2 -450.662} C_VEL
LIN {X 0,Y 608.444,Z 709.191,A -85,B 0,C 180,E1 -451.986,E2 -451.986} C_VEL
LIN {X 0,Y 608.421,Z 706.885,A -85,B 0,C 180,E1 -453.311,E2 -453.311} C_VEL
LIN {X 0,Y 608.427,Z 703.383,A -85,B 0,C 180,E1 -454.638,E2 -454.638} C_VEL
LIN {X 0,Y 608.435,Z 698.608,A -85,B 0,C 180,E1 -455.967,E2 -455.967} C_VEL
LIN {X 0,Y 608.456,Z 692.426,A -85,B 0,C 180,E1 -457.299,E2 -457.299} C_VEL
LIN {X 0,Y 608.464,Z 684.654,A -85,B 0,C 180,E1 -458.636,E2 -458.636} C_VEL
LIN {X 0,Y 608.471,Z 676.37,A -85,B 0,C 180,E1 -459.809,E2 -459.809} C_VEL
LIN {X 0,Y 608.492,Z 665.652,A -85,B 0,C 180,E1 -461.063,E2 -461.063} C_VEL
LIN {X 0,Y 608.523,Z 654.274,A -85,B 0,C 180,E1 -462.168,E2 -462.168} C_VEL
LIN {X 0,Y 608.547,Z 642.854,A -85,B 0,C 180,E1 -463.1,E2 -463.1} C_VEL
LIN {X 0,Y 608.563,Z 630.446,A -85,B 0,C 180,E1 -463.95,E2 -463.95} C_VEL
LIN {X 0,Y 608.56,Z 616.858,A -85,B 0,C 180,E1 -464.718,E2 -464.718} C_VEL
LIN {X 0,Y 608.631,Z 602.79,A -85,B 0,C 180,E1 -465.359,E2 -465.359} C_VEL
LIN {X 0,Y 608.635,Z 588.3,A -85,B 0,C 180,E1 -465.874,E2 -465.874} C_VEL
LIN {X 0,Y 608.682,Z 573.042,A -85,B 0,C 180,E1 -466.269,E2 -466.269} C_VEL
LIN {X 0,Y 608.682,Z 557.166,A -85,B 0,C 180,E1 -466.533,E2 -466.533} C_VEL
LIN {X 0,Y 608.685,Z 399.645,A -85,B 0,C 180,E1 -468.442,E2 -468.442} C_VEL
LIN {X 0,Y 608.543,Z 398.536,A -85,B 0,C 180,E1 -468.495,E2 -468.495} C_VEL
LIN {X 0,Y 608.619,Z 373.248,A -85,B 0,C 180,E1 -471.33,E2 -471.33} C_VEL
LIN {X 0,Y 608.685,Z 347.17,A -85,B 0,C 180,E1 -474.313,E2 -474.313} C_VEL
LIN {X 0,Y 608.424,Z 338.318,A -85,B 0,C 180,E1 -475.356,E2 -475.356} C_VEL
LIN {X 0,Y 608.45,Z 338.323,A -85,B 0,C 180,E1 -478.267,E2 -478.267} C_VEL
LIN {X 0,Y 608.455,Z 338.319,A -85,B 0,C 180,E1 -480.546,E2 -480.546} C_VEL
LIN {X 0,Y 608.434,Z 338.317,A -85,B 0,C 180,E1 -482.881,E2 -482.881} C_VEL
LIN {X 0,Y 608.415,Z 338.317,A -85,B 0,C 180,E1 -485.28,E2 -485.28} C_VEL
LIN {X 0,Y 608.464,Z 338.319,A -85,B 0,C 180,E1 -488.24,E2 -488.24} C_VEL
LIN {X 0,Y 608.41,Z 338.318,A -85,B 0,C 180,E1 -491.18,E2 -491.18} C_VEL
LIN {X 0,Y 608.432,Z 338.315,A -85,B 0,C 180,E1 -493.305,E2 -493.305} C_VEL
LIN {X 0,Y 608.467,Z 338.317,A -85,B 0,C 180,E1 -496.131,E2 -496.131} C_VEL
LIN {X 0,Y 608.423,Z 338.319,A -85,B 0,C 180,E1 -498.821,E2 -498.821} C_VEL
LIN {X 0,Y 608.457,Z 338.313,A -85,B 0,C 180,E1 -501.761,E2 -501.761} C_VEL
LIN {X 0,Y 608.433,Z 338.32,A -85,B 0,C 180,E1 -504.722,E2 -504.722} C_VEL
LIN {X 0,Y 608.432,Z 338.315,A -85,B 0,C 180,E1 -507.119,E2 -507.119} C_VEL
LIN {X 0,Y 608.471,Z 338.314,A -85,B 0,C 180,E1 -510.028,E2 -510.028} C_VEL
LIN {X 0,Y 608.453,Z 338.316,A -85,B 0,C 180,E1 -512.798,E2 -512.798} C_VEL
LIN {X 0,Y 608.43,Z 338.315,A -85,B 0,C 180,E1 -515.428,E2 -515.428} C_VEL
LIN {X 0,Y 608.465,Z 338.32,A -85,B 0,C 180,E1 -518.309,E2 -518.309} C_VEL
LIN {X 0,Y 608.436,Z 338.315,A -85,B 0,C 180,E1 -521.13,E2 -521.13} C_VEL
LIN {X 0,Y 608.454,Z 338.314,A -85,B 0,C 180,E1 -523.906,E2 -523.906} C_VEL
LIN {X 0,Y 608.447,Z 338.32,A -85,B 0,C 180,E1 -526.643,E2 -526.643} C_VEL
LIN {X 0,Y 608.428,Z 338.315,A -85,B 0,C 180,E1 -529.35,E2 -529.35} C_VEL
LIN {X 0,Y 608.48,Z 338.312,A -85,B 0,C 180,E1 -532.033,E2 -532.033} C_VEL
LIN {X 0,Y 608.448,Z 338.319,A -85,B 0,C 180,E1 -534.698,E2 -534.698} C_VEL
LIN {X 0,Y 608.442,Z 338.313,A -85,B 0,C 180,E1 -537.352,E2 -537.352} C_VEL
LIN {X 0,Y 608.477,Z 338.312,A -85,B 0,C 180,E1 -540,E2 -540} C_VEL
LIN {X 0,Y 608.471,Z 338.317,A -85,B 0,C 180,E1 -542.648,E2 -542.648} C_VEL
LIN {X 0,Y 608.431,Z 338.315,A -85,B 0,C 180,E1 -545.302,E2 -545.302} C_VEL
LIN {X 0,Y 608.475,Z 338.312,A -85,B 0,C 180,E1 -547.967,E2 -547.967} C_VEL
LIN {X 0,Y 608.435,Z 338.314,A -85,B 0,C 180,E1 -549.456,E2 -549.456} C_VEL
LIN {X 0,Y 607.773,Z 338.401,A -85,B 0,C 180,E1 -550.008,E2 -550.008} C_VEL
LIN {X 0,Y 604.932,Z 338.754,A -85,B 0,C 180,E1 -550.905,E2 -550.905} C_VEL
LIN {X 0,Y 602.527,Z 339.055,A -85,B 0,C 180,E1 -551.627,E2 -551.627} C_VEL
LIN {X 0,Y 601.49,Z 339.185,A -85,B 0,C 180,E1 -552.183,E2 -552.183} C_VEL
LIN {X 0,Y 601.403,Z 339.194,A -85,B 0,C 180,E1 -552.372,E2 -552.372} C_VEL
LIN {X 0,Y 601.419,Z 339.192,A -85,B 0,C 180,E1 -554.898,E2 -554.898} C_VEL
LIN {X 0,Y 601.407,Z 339.193,A -85,B 0,C 180,E1 -556.987,E2 -556.987} C_VEL
LIN {X 0,Y 601.41,Z 339.19,A -85,B 0,C 180,E1 -559.1,E2 -559.1} C_VEL
LIN {X 0,Y 601.393,Z 339.192,A -85,B 0,C 180,E1 -561.24,E2 -561.24} C_VEL
LIN {X 0,Y 601.463,Z 339.187,A -85,B 0,C 180,E1 -564.141,E2 -564.141} C_VEL
LIN {X 0,Y 601.392,Z 339.193,A -85,B 0,C 180,E1 -567.114,E2 -567.114} C_VEL
LIN {X 0,Y 601.395,Z 339.191,A -85,B 0,C 180,E1 -569.395,E2 -569.395} C_VEL
LIN {X 0,Y 601.399,Z 339.191,A -85,B 0,C 180,E1 -571.728,E2 -571.728} C_VEL
LIN {X 0,Y 601.422,Z 339.192,A -85,B 0,C 180,E1 -574.119,E2 -574.119} C_VEL
LIN {X 0,Y 601.392,Z 339.202,A -85,B 0,C 180,E1 -576.584,E2 -576.584} C_VEL
LIN {X 0,Y 601.391,Z 339.193,A -85,B 0,C 180,E1 -579.129,E2 -579.129} C_VEL
LIN {X 0,Y 601.421,Z 339.189,A -85,B 0,C 180,E1 -581.766,E2 -581.766} C_VEL
LIN {X 0,Y 601.402,Z 339.202,A -85,B 0,C 180,E1 -584.533,E2 -584.533} C_VEL
LIN {X 0,Y 601.433,Z 339.195,A -85,B 0,C 180,E1 -586.428,E2 -586.428} C_VEL
LIN {X 0,Y 601.405,Z 339.192,A -85,B 0,C 180,E1 -589.125,E2 -589.125} C_VEL
LIN {X 0,Y 601.41,Z 339.19,A -85,B 0,C 180,E1 -591.731,E2 -591.731} C_VEL
LIN {X 0,Y 601.389,Z 339.198,A -85,B 0,C 180,E1 -594.245,E2 -594.245} C_VEL
LIN {X 0,Y 601.426,Z 339.198,A -85,B 0,C 180,E1 -596.686,E2 -596.686} C_VEL
LIN {X 0,Y 601.431,Z 339.31,A -85,B 0,C 180,E1 -597.559,E2 -597.559} C_VEL
LIN {X 0,Y 601.653,Z 344.666,A -85,B 0,C 180,E1 -598.288,E2 -598.288} C_VEL
LIN {X 0,Y 601.592,Z 364.647,A -85,B 0,C 180,E1 -600.943,E2 -600.943} C_VEL
LIN {X 0,Y 601.567,Z 367.973,A -85,B 0,C 180,E1 -601.38,E2 -601.38} C_VEL
LIN {X 0,Y 602.022,Z 371.233,A -85,B 0,C 180,E1 -601.436,E2 -601.436} C_VEL
LIN {X 0,Y 601.873,Z 532.501,A -85,B 0,C 180,E1 -603.425,E2 -603.425} C_VEL
LIN {X 0,Y 601.832,Z 548.146,A -85,B 0,C 180,E1 -603.755,E2 -603.755} C_VEL
LIN {X 0,Y 601.774,Z 563.452,A -85,B 0,C 180,E1 -604.225,E2 -604.225} C_VEL
LIN {X 0,Y 601.709,Z 577.829,A -85,B 0,C 180,E1 -604.812,E2 -604.812} C_VEL
LIN {X 0,Y 601.65,Z 591.769,A -85,B 0,C 180,E1 -605.529,E2 -605.529} C_VEL
LIN {X 0,Y 601.58,Z 605.73,A -85,B 0,C 180,E1 -606.414,E2 -606.414} C_VEL
LIN {X 0,Y 601.539,Z 618.113,A -85,B 0,C 180,E1 -607.368,E2 -607.368} C_VEL
LIN {X 0,Y 601.459,Z 629.376,A -85,B 0,C 180,E1 -608.403,E2 -608.403} C_VEL
LIN {X 0,Y 601.445,Z 639.217,A -85,B 0,C 180,E1 -609.479,E2 -609.479} C_VEL
LIN {X 0,Y 601.409,Z 648.777,A -85,B 0,C 180,E1 -610.724,E2 -610.724} C_VEL
LIN {X 0,Y 601.385,Z 656.609,A -85,B 0,C 180,E1 -611.96,E2 -611.96} C_VEL
LIN {X 0,Y 601.372,Z 662.163,A -85,B 0,C 180,E1 -613.012,E2 -613.012} C_VEL
LIN {X 0,Y 601.336,Z 668.156,A -85,B 0,C 180,E1 -614.407,E2 -614.407} C_VEL
LIN {X 0,Y 601.328,Z 672.676,A -85,B 0,C 180,E1 -615.792,E2 -615.792} C_VEL
LIN {X 0,Y 601.323,Z 675.862,A -85,B 0,C 180,E1 -617.17,E2 -617.17} C_VEL
LIN {X 0,Y 601.323,Z 677.778,A -85,B 0,C 180,E1 -618.54,E2 -618.54} C_VEL
LIN {X 0,Y 601.325,Z 678.473,A -85,B 0,C 180,E1 -619.903,E2 -619.903} C_VEL
LIN {X 0,Y 601.327,Z 677.999,A -85,B 0,C 180,E1 -621.261,E2 -621.261} C_VEL
LIN {X 0,Y 601.319,Z 676.368,A -85,B 0,C 180,E1 -622.613,E2 -622.613} C_VEL
LIN {X 0,Y 601.33,Z 673.563,A -85,B 0,C 180,E1 -623.962,E2 -623.962} C_VEL
LIN {X 0,Y 601.332,Z 669.539,A -85,B 0,C 180,E1 -625.307,E2 -625.307} C_VEL
LIN {X 0,Y 601.349,Z 664.205,A -85,B 0,C 180,E1 -626.65,E2 -626.65} C_VEL
LIN {X 0,Y 601.382,Z 657.417,A -85,B 0,C 180,E1 -627.991,E2 -627.991} C_VEL
LIN {X 0,Y 601.411,Z 649.029,A -85,B 0,C 180,E1 -629.33,E2 -629.33} C_VEL
LIN {X 0,Y 601.441,Z 640.123,A -85,B 0,C 180,E1 -630.502,E2 -630.502} C_VEL
LIN {X 0,Y 601.481,Z 629.5,A -85,B 0,C 180,E1 -631.674,E2 -631.674} C_VEL
LIN {X 0,Y 601.53,Z 617.622,A -85,B 0,C 180,E1 -632.762,E2 -632.762} C_VEL
LIN {X 0,Y 601.587,Z 605.612,A -85,B 0,C 180,E1 -633.684,E2 -633.684} C_VEL
LIN {X 0,Y 601.657,Z 592.459,A -85,B 0,C 180,E1 -634.522,E2 -634.522} C_VEL
LIN {X 0,Y 601.71,Z 577.844,A -85,B 0,C 180,E1 -635.278,E2 -635.278} C_VEL
LIN {X 0,Y 601.787,Z 563.441,A -85,B 0,C 180,E1 -635.865,E2 -635.865} C_VEL
LIN {X 0,Y 601.829,Z 547.557,A -85,B 0,C 180,E1 -636.35,E2 -636.35} C_VEL
LIN {X 0,Y 601.865,Z 532.706,A -85,B 0,C 180,E1 -636.662,E2 -636.662} C_VEL
LIN {X 0,Y 602.011,Z 370.318,A -85,B 0,C 180,E1 -638.666,E2 -638.666} C_VEL
LIN {X 0,Y 601.604,Z 367.772,A -85,B 0,C 180,E1 -638.735,E2 -638.735} C_VEL
LIN {X 0,Y 601.652,Z 347.265,A -85,B 0,C 180,E1 -641.454,E2 -641.454} C_VEL
LIN {X 0,Y 601.477,Z 339.648,A -85,B 0,C 180,E1 -642.484,E2 -642.484} C_VEL
LIN {X 0,Y 601.394,Z 339.196,A -85,B 0,C 180,E1 -642.571,E2 -642.571} C_VEL
LIN {X 0,Y 601.392,Z 339.194,A -85,B 0,C 180,E1 -644.898,E2 -644.898} C_VEL
LIN {X 0,Y 601.405,Z 339.193,A -85,B 0,C 180,E1 -646.987,E2 -646.987} C_VEL
LIN {X 0,Y 601.399,Z 339.197,A -85,B 0,C 180,E1 -649.81,E2 -649.81} C_VEL
LIN {X 0,Y 601.404,Z 339.19,A -85,B 0,C 180,E1 -652.683,E2 -652.683} C_VEL
LIN {X 0,Y 601.388,Z 339.194,A -85,B 0,C 180,E1 -654.879,E2 -654.879} C_VEL
LIN {X 0,Y 601.403,Z 339.198,A -85,B 0,C 180,E1 -657.359,E2 -657.359} C_VEL
LIN {X 0,Y 601.41,Z 339.191,A -85,B 0,C 180,E1 -660.165,E2 -660.165} C_VEL
LIN {X 0,Y 601.401,Z 339.19,A -85,B 0,C 180,E1 -662.711,E2 -662.711} C_VEL
LIN {X 0,Y 601.378,Z 339.197,A -85,B 0,C 180,E1 -665.109,E2 -665.109} C_VEL
LIN {X 0,Y 601.405,Z 339.198,A -85,B 0,C 180,E1 -667.421,E2 -667.421} C_VEL
LIN {X 0,Y 601.403,Z 339.193,A -85,B 0,C 180,E1 -669.996,E2 -669.996} C_VEL
LIN {X 0,Y 601.372,Z 339.194,A -85,B 0,C 180,E1 -672.674,E2 -672.674} C_VEL
LIN {X 0,Y 601.403,Z 339.2,A -85,B 0,C 180,E1 -675.479,E2 -675.479} C_VEL
LIN {X 0,Y 601.409,Z 339.19,A -85,B 0,C 180,E1 -678.409,E2 -678.409} C_VEL
LIN {X 0,Y 601.387,Z 339.193,A -85,B 0,C 180,E1 -680.871,E2 -680.871} C_VEL
LIN {X 0,Y 601.396,Z 339.199,A -85,B 0,C 180,E1 -683.741,E2 -683.741} C_VEL
LIN {X 0,Y 601.411,Z 339.189,A -85,B 0,C 180,E1 -686.685,E2 -686.685} C_VEL
LIN {X 0,Y 601.403,Z 339.193,A -85,B 0,C 180,E1 -689.057,E2 -689.057} C_VEL
LIN {X 0,Y 601.427,Z 339.194,A -85,B 0,C 180,E1 -691.372,E2 -691.372} C_VEL
LIN {X 0,Y 601.396,Z 339.19,A -85,B 0,C 180,E1 -694.38,E2 -694.38} C_VEL
LIN {X 0,Y 601.381,Z 339.192,A -85,B 0,C 180,E1 -696.588,E2 -696.588} C_VEL
LIN {X 0,Y 601.428,Z 339.196,A -85,B 0,C 180,E1 -699.478,E2 -699.478} C_VEL
LIN {X 0,Y 601.381,Z 339.193,A -85,B 0,C 180,E1 -702.311,E2 -702.311} C_VEL
LIN {X 0,Y 601.393,Z 339.192,A -85,B 0,C 180,E1 -704.408,E2 -704.408} C_VEL
LIN {X 0,Y 601.402,Z 339.194,A -85,B 0,C 180,E1 -707.171,E2 -707.171} C_VEL
LIN {X 0,Y 601.428,Z 339.192,A -85,B 0,C 180,E1 -709.905,E2 -709.905} C_VEL
LIN {X 0,Y 601.378,Z 339.193,A -85,B 0,C 180,E1 -712.614,E2 -712.614} C_VEL
LIN {X 0,Y 601.406,Z 339.195,A -85,B 0,C 180,E1 -715.308,E2 -715.308} C_VEL
LIN {X 0,Y 601.433,Z 339.191,A -85,B 0,C 180,E1 -717.991,E2 -717.991} C_VEL
LIN {X 0,Y 601.396,Z 339.191,A -85,B 0,C 180,E1 -720.669,E2 -720.669} C_VEL
LIN {X 0,Y 601.411,Z 339.195,A -85,B 0,C 180,E1 -723.349,E2 -723.349} C_VEL
LIN {X 0,Y 601.413,Z 339.192,A -85,B 0,C 180,E1 -726.037,E2 -726.037} C_VEL
LIN {X 0,Y 601.387,Z 339.192,A -85,B 0,C 180,E1 -728.738,E2 -728.738} C_VEL
LIN {X 0,Y 601.409,Z 339.198,A -85,B 0,C 180,E1 -731.458,E2 -731.458} C_VEL
LIN {X 0,Y 601.415,Z 339.19,A -85,B 0,C 180,E1 -734.205,E2 -734.205} C_VEL
LIN {X 0,Y 601.378,Z 339.195,A -85,B 0,C 180,E1 -736.987,E2 -736.987} C_VEL
LIN {X 0,Y 601.394,Z 339.199,A -85,B 0,C 180,E1 -739.81,E2 -739.81} C_VEL
LIN {X 0,Y 601.4,Z 339.19,A -85,B 0,C 180,E1 -742.683,E2 -742.683} C_VEL
LIN {X 0,Y 601.383,Z 339.193,A -85,B 0,C 180,E1 -744.879,E2 -744.879} C_VEL
LIN {X 0,Y 601.397,Z 339.197,A -85,B 0,C 180,E1 -747.358,E2 -747.358} C_VEL
LIN {X 0,Y 601.406,Z 339.192,A -85,B 0,C 180,E1 -750.165,E2 -750.165} C_VEL
LIN {X 0,Y 601.396,Z 339.191,A -85,B 0,C 180,E1 -752.711,E2 -752.711} C_VEL
LIN {X 0,Y 601.374,Z 339.196,A -85,B 0,C 180,E1 -755.109,E2 -755.109} C_VEL
LIN {X 0,Y 601.399,Z 339.198,A -85,B 0,C 180,E1 -757.422,E2 -757.422} C_VEL
LIN {X 0,Y 601.4,Z 339.195,A -85,B 0,C 180,E1 -759.996,E2 -759.996} C_VEL
LIN {X 0,Y 601.365,Z 339.195,A -85,B 0,C 180,E1 -762.674,E2 -762.674} C_VEL
LIN {X 0,Y 601.399,Z 339.199,A -85,B 0,C 180,E1 -765.479,E2 -765.479} C_VEL
LIN {X 0,Y 601.406,Z 339.191,A -85,B 0,C 180,E1 -768.409,E2 -768.409} C_VEL
LIN {X 0,Y 601.382,Z 339.194,A -85,B 0,C 180,E1 -770.871,E2 -770.871} C_VEL
LIN {X 0,Y 601.392,Z 339.201,A -85,B 0,C 180,E1 -773.741,E2 -773.741} C_VEL
LIN {X 0,Y 601.407,Z 339.19,A -85,B 0,C 180,E1 -776.685,E2 -776.685} C_VEL
LIN {X 0,Y 601.399,Z 339.193,A -85,B 0,C 180,E1 -779.057,E2 -779.057} C_VEL
LIN {X 0,Y 601.418,Z 339.195,A -85,B 0,C 180,E1 -781.372,E2 -781.372} C_VEL
LIN {X 0,Y 601.396,Z 339.195,A -85,B 0,C 180,E1 -784.427,E2 -784.427} C_VEL
LIN {X 0,Y 601.84,Z 343.461,A -85,B 0,C 180,E1 -784.956,E2 -784.956} C_VEL
LIN {X 0,Y 601.771,Z 365.894,A -85,B 0,C 180,E1 -787.568,E2 -787.568} C_VEL
LIN {X 0,Y 601.684,Z 390.492,A -85,B 0,C 180,E1 -790.378,E2 -790.378} C_VEL
LIN {X 0,Y 601.628,Z 398.844,A -85,B 0,C 180,E1 -791.32,E2 -791.32} C_VEL
LIN {X 0,Y 602.027,Z 403.039,A -85,B 0,C 180,E1 -791.389,E2 -791.389} C_VEL
LIN {X 0,Y 601.886,Z 564.282,A -85,B 0,C 180,E1 -793.377,E2 -793.377} C_VEL
LIN {X 0,Y 601.86,Z 579.884,A -85,B 0,C 180,E1 -793.704,E2 -793.704} C_VEL
LIN {X 0,Y 601.786,Z 594.789,A -85,B 0,C 180,E1 -794.158,E2 -794.158} C_VEL
LIN {X 0,Y 601.72,Z 609.757,A -85,B 0,C 180,E1 -794.764,E2 -794.764} C_VEL
LIN {X 0,Y 601.658,Z 623.231,A -85,B 0,C 180,E1 -795.455,E2 -795.455} C_VEL
LIN {X 0,Y 601.617,Z 636.448,A -85,B 0,C 180,E1 -796.283,E2 -796.283} C_VEL
LIN {X 0,Y 601.531,Z 648.283,A -85,B 0,C 180,E1 -797.174,E2 -797.174} C_VEL
LIN {X 0,Y 601.489,Z 659.747,A -85,B 0,C 180,E1 -798.201,E2 -798.201} C_VEL
LIN {X 0,Y 601.43,Z 669.388,A -85,B 0,C 180,E1 -799.224,E2 -799.224} C_VEL
LIN {X 0,Y 601.428,Z 678.854,A -85,B 0,C 180,E1 -800.414,E2 -800.414} C_VEL
LIN {X 0,Y 601.369,Z 686.73,A -85,B 0,C 180,E1 -801.6,E2 -801.6} C_VEL
LIN {X 0,Y 601.367,Z 694.087,A -85,B 0,C 180,E1 -802.951,E2 -802.951} C_VEL
LIN {X 0,Y 601.373,Z 699.924,A -85,B 0,C 180,E1 -804.299,E2 -804.299} C_VEL
LIN {X 0,Y 601.329,Z 703.383,A -85,B 0,C 180,E1 -805.307,E2 -805.307} C_VEL
LIN {X 0,Y 601.338,Z 706.886,A -85,B 0,C 180,E1 -806.65,E2 -806.65} C_VEL
LIN {X 0,Y 601.342,Z 709.192,A -85,B 0,C 180,E1 -807.991,E2 -807.991} C_VEL
LIN {X 0,Y 601.335,Z 710.35,A -85,B 0,C 180,E1 -809.33,E2 -809.33} C_VEL
LIN {X 0,Y 601.335,Z 710.35,A -85,B 0,C 180,E1 -810.67,E2 -810.67} C_VEL
LIN {X 0,Y 601.342,Z 709.192,A -85,B 0,C 180,E1 -812.009,E2 -812.009} C_VEL
LIN {X 0,Y 601.337,Z 706.886,A -85,B 0,C 180,E1 -813.35,E2 -813.35} C_VEL
LIN {X 0,Y 601.329,Z 703.383,A -85,B 0,C 180,E1 -814.693,E2 -814.693} C_VEL
LIN {X 0,Y 601.356,Z 698.608,A -85,B 0,C 180,E1 -816.038,E2 -816.038} C_VEL
LIN {X 0,Y 601.365,Z 692.425,A -85,B 0,C 180,E1 -817.386,E2 -817.386} C_VEL
LIN {X 0,Y 601.386,Z 684.653,A -85,B 0,C 180,E1 -818.738,E2 -818.738} C_VEL
LIN {X 0,Y 601.428,Z 676.37,A -85,B 0,C 180,E1 -819.925,E2 -819.925} C_VEL
LIN {X 0,Y 601.46,Z 665.932,A -85,B 0,C 180,E1 -821.165,E2 -821.165} C_VEL
LIN {X 0,Y 601.514,Z 656.192,A -85,B 0,C 180,E1 -822.14,E2 -822.14} C_VEL
LIN {X 0,Y 601.57,Z 644.015,A -85,B 0,C 180,E1 -823.168,E2 -823.168} C_VEL
LIN {X 0,Y 601.606,Z 632.077,A -85,B 0,C 180,E1 -824.012,E2 -824.012} C_VEL
LIN {X 0,Y 601.65,Z 618.526,A -85,B 0,C 180,E1 -824.805,E2 -824.805} C_VEL
LIN {X 0,Y 601.763,Z 603.842,A -85,B 0,C 180,E1 -825.495,E2 -825.495} C_VEL
LIN {X 0,Y 601.786,Z 589.617,A -85,B 0,C 180,E1 -826.016,E2 -826.016} C_VEL
LIN {X 0,Y 601.853,Z 574.718,A -85,B 0,C 180,E1 -826.419,E2 -826.419} C_VEL
LIN {X 0,Y 601.866,Z 559.746,A -85,B 0,C 180,E1 -826.689,E2 -826.689} C_VEL
LIN {X 0,Y 601.906,Z 400.45,A -85,B 0,C 180,E1 -828.647,E2 -828.647} C_VEL
LIN {X 0,Y 601.629,Z 398.715,A -85,B 0,C 180,E1 -828.695,E2 -828.695} C_VEL
LIN {X 0,Y 601.748,Z 373.248,A -85,B 0,C 180,E1 -831.586,E2 -831.586} C_VEL
LIN {X 0,Y 601.879,Z 349.049,A -85,B 0,C 180,E1 -834.386,E2 -834.386} C_VEL
LIN {X 0,Y 601.636,Z 340.326,A -85,B 0,C 180,E1 -835.423,E2 -835.423} C_VEL
LIN {X 0,Y 601.395,Z 339.197,A -85,B 0,C 180,E1 -835.573,E2 -835.573} C_VEL
LIN {X 0,Y 601.418,Z 339.195,A -85,B 0,C 180,E1 -838.628,E2 -838.628} C_VEL
LIN {X 0,Y 601.409,Z 339.19,A -85,B 0,C 180,E1 -841.453,E2 -841.453} C_VEL
LIN {X 0,Y 601.414,Z 339.196,A -85,B 0,C 180,E1 -844.119,E2 -844.119} C_VEL
LIN {X 0,Y 601.381,Z 339.2,A -85,B 0,C 180,E1 -846.585,E2 -846.585} C_VEL
LIN {X 0,Y 601.382,Z 339.193,A -85,B 0,C 180,E1 -849.129,E2 -849.129} C_VEL
LIN {X 0,Y 601.417,Z 339.19,A -85,B 0,C 180,E1 -851.766,E2 -851.766} C_VEL
LIN {X 0,Y 601.397,Z 339.199,A -85,B 0,C 180,E1 -854.533,E2 -854.533} C_VEL
LIN {X 0,Y 601.371,Z 339.194,A -85,B 0,C 180,E1 -857.414,E2 -857.414} C_VEL
LIN {X 0,Y 601.4,Z 339.195,A -85,B 0,C 180,E1 -860.004,E2 -860.004} C_VEL
LIN {X 0,Y 601.399,Z 339.197,A -85,B 0,C 180,E1 -862.623,E2 -862.623} C_VEL
LIN {X 0,Y 601.379,Z 339.194,A -85,B 0,C 180,E1 -865.066,E2 -865.066} C_VEL
LIN {X 0,Y 601.404,Z 339.19,A -85,B 0,C 180,E1 -867.483,E2 -867.483} C_VEL
LIN {X 0,Y 601.408,Z 339.191,A -85,B 0,C 180,E1 -869.855,E2 -869.855} C_VEL
LIN {X 0,Y 601.399,Z 339.197,A -85,B 0,C 180,E1 -872.641,E2 -872.641} C_VEL
LIN {X 0,Y 601.385,Z 339.193,A -85,B 0,C 180,E1 -875.121,E2 -875.121} C_VEL
LIN {X 0,Y 601.397,Z 339.195,A -85,B 0,C 180,E1 -878.04,E2 -878.04} C_VEL
LIN {X 0,Y 601.407,Z 339.193,A -85,B 0,C 180,E1 -880.901,E2 -880.901} C_VEL
LIN {X 0,Y 601.413,Z 339.19,A -85,B 0,C 180,E1 -883.713,E2 -883.713} C_VEL
LIN {X 0,Y 601.407,Z 339.2,A -85,B 0,C 180,E1 -886.484,E2 -886.484} C_VEL
LIN {X 0,Y 601.387,Z 339.193,A -85,B 0,C 180,E1 -889.224,E2 -889.224} C_VEL
LIN {X 0,Y 601.439,Z 339.188,A -85,B 0,C 180,E1 -891.939,E2 -891.939} C_VEL
LIN {X 0,Y 601.415,Z 339.196,A -85,B 0,C 180,E1 -894.636,E2 -894.636} C_VEL
LIN {X 0,Y 601.412,Z 339.189,A -85,B 0,C 180,E1 -897.321,E2 -897.321} C_VEL
LIN {X 0,Y 601.445,Z 339.188,A -85,B 0,C 180,E1 -900,E2 -900} C_VEL
LIN {X 0,Y 601.434,Z 339.193,A -85,B 0,C 180,E1 -902.679,E2 -902.679} C_VEL
LIN {X 0,Y 601.399,Z 339.191,A -85,B 0,C 180,E1 -905.365,E2 -905.365} C_VEL
LIN {X 0,Y 601.438,Z 339.189,A -85,B 0,C 180,E1 -908.061,E2 -908.061} C_VEL
LIN {X 0,Y 601.401,Z 339.193,A -85,B 0,C 180,E1 -910.999,E2 -910.999} C_VEL
LIN {X 0,Y 601.403,Z 339.194,A -85,B 0,C 180,E1 -912.372,E2 -912.372} C_VEL
LIN {X 0,Y 600.732,Z 339.278,A -85,B 0,C 180,E1 -912.931,E2 -912.931} C_VEL
LIN {X 0,Y 597.881,Z 339.632,A -85,B 0,C 180,E1 -913.839,E2 -913.839} C_VEL
LIN {X 0,Y 595.473,Z 339.938,A -85,B 0,C 180,E1 -914.569,E2 -914.569} C_VEL
LIN {X 0,Y 594.436,Z 340.06,A -85,B 0,C 180,E1 -915.133,E2 -915.133} C_VEL
LIN {X 0,Y 594.349,Z 340.069,A -85,B 0,C 180,E1 -915.324,E2 -915.324} C_VEL
LIN {X 0,Y 594.373,Z 340.067,A -85,B 0,C 180,E1 -917.194,E2 -917.194} C_VEL
LIN {X 0,Y 594.37,Z 340.068,A -85,B 0,C 180,E1 -920.054,E2 -920.054} C_VEL
LIN {X 0,Y 594.355,Z 340.071,A -85,B 0,C 180,E1 -922.968,E2 -922.968} C_VEL
LIN {X 0,Y 594.354,Z 340.068,A -85,B 0,C 180,E1 -925.194,E2 -925.194} C_VEL
LIN {X 0,Y 594.374,Z 340.072,A -85,B 0,C 180,E1 -928.228,E2 -928.228} C_VEL
LIN {X 0,Y 594.379,Z 340.074,A -85,B 0,C 180,E1 -930.56,E2 -930.56} C_VEL
LIN {X 0,Y 594.379,Z 340.069,A -85,B 0,C 180,E1 -932.951,E2 -932.951} C_VEL
LIN {X 0,Y 594.328,Z 340.071,A -85,B 0,C 180,E1 -935.411,E2 -935.411} C_VEL
LIN {X 0,Y 594.375,Z 340.068,A -85,B 0,C 180,E1 -937.942,E2 -937.942} C_VEL
LIN {X 0,Y 594.367,Z 340.073,A -85,B 0,C 180,E1 -940.821,E2 -940.821} C_VEL
LIN {X 0,Y 594.353,Z 340.069,A -85,B 0,C 180,E1 -943.301,E2 -943.301} C_VEL
LIN {X 0,Y 594.364,Z 340.071,A -85,B 0,C 180,E1 -946.162,E2 -946.162} C_VEL
LIN {X 0,Y 594.381,Z 340.076,A -85,B 0,C 180,E1 -948.536,E2 -948.536} C_VEL
LIN {X 0,Y 594.37,Z 340.068,A -85,B 0,C 180,E1 -951.298,E2 -951.298} C_VEL
LIN {X 0,Y 594.35,Z 340.07,A -85,B 0,C 180,E1 -953.755,E2 -953.755} C_VEL
LIN {X 0,Y 594.381,Z 340.072,A -85,B 0,C 180,E1 -956.239,E2 -956.239} C_VEL
LIN {X 0,Y 594.408,Z 340.232,A -85,B 0,C 180,E1 -957.404,E2 -957.404} C_VEL
LIN {X 0,Y 594.77,Z 343.595,A -85,B 0,C 180,E1 -957.877,E2 -957.877} C_VEL
LIN {X 0,Y 594.641,Z 364.027,A -85,B 0,C 180,E1 -960.628,E2 -960.628} C_VEL
LIN {X 0,Y 594.648,Z 367.911,A -85,B 0,C 180,E1 -961.147,E2 -961.147} C_VEL
LIN {X 0,Y 595.307,Z 372.232,A -85,B 0,C 180,E1 -961.231,E2 -961.231} C_VEL
LIN {X 0,Y 595.068,Z 533.108,A -85,B 0,C 180,E1 -963.239,E2 -963.239} C_VEL
LIN {X 0,Y 595.02,Z 548.72,A -85,B 0,C 180,E1 -963.578,E2 -963.578} C_VEL
LIN {X 0,Y 594.94,Z 563.093,A -85,B 0,C 180,E1 -964.026,E2 -964.026} C_VEL
LIN {X 0,Y 594.838,Z 578.037,A -85,B 0,C 180,E1 -964.641,E2 -964.641} C_VEL
LIN {X 0,Y 594.734,Z 592.57,A -85,B 0,C 180,E1 -965.402,E2 -965.402} C_VEL
LIN {X 0,Y 594.637,Z 605.184,A -85,B 0,C 180,E1 -966.214,E2 -966.214} C_VEL
LIN {X 0,Y 594.553,Z 618.195,A -85,B 0,C 180,E1 -967.223,E2 -967.223} C_VEL
LIN {X 0,Y 594.443,Z 629.89,A -85,B 0,C 180,E1 -968.317,E2 -968.317} C_VEL
LIN {X 0,Y 594.394,Z 639.666,A -85,B 0,C 180,E1 -969.405,E2 -969.405} C_VEL
LIN {X 0,Y 594.346,Z 649.14,A -85,B 0,C 180,E1 -970.665,E2 -970.665} C_VEL
LIN {X 0,Y 594.304,Z 656.919,A -85,B 0,C 180,E1 -971.915,E2 -971.915} C_VEL
LIN {X 0,Y 594.274,Z 664.026,A -85,B 0,C 180,E1 -973.322,E2 -973.322} C_VEL
LIN {X 0,Y 594.261,Z 668.987,A -85,B 0,C 180,E1 -974.568,E2 -974.568} C_VEL
LIN {X 0,Y 594.265,Z 673.028,A -85,B 0,C 180,E1 -975.876,E2 -975.876} C_VEL
LIN {X 0,Y 594.242,Z 675.644,A -85,B 0,C 180,E1 -977.014,E2 -977.014} C_VEL
LIN {X 0,Y 594.234,Z 677.641,A -85,B 0,C 180,E1 -978.401,E2 -978.401} C_VEL
LIN {X 0,Y 594.227,Z 678.446,A -85,B 0,C 180,E1 -979.781,E2 -979.781} C_VEL
LIN {X 0,Y 594.223,Z 678.082,A -85,B 0,C 180,E1 -981.155,E2 -981.155} C_VEL
LIN {X 0,Y 594.223,Z 676.563,A -85,B 0,C 180,E1 -982.525,E2 -982.525} C_VEL
LIN {X 0,Y 594.235,Z 673.875,A -85,B 0,C 180,E1 -983.89,E2 -983.89} C_VEL
LIN {X 0,Y 594.236,Z 669.956,A -85,B 0,C 180,E1 -985.251,E2 -985.251} C_VEL
LIN {X 0,Y 594.271,Z 664.707,A -85,B 0,C 180,E1 -986.61,E2 -986.61} C_VEL
LIN {X 0,Y 594.296,Z 658.051,A -85,B 0,C 180,E1 -987.967,E2 -987.967} C_VEL
LIN {X 0,Y 594.333,Z 650.921,A -85,B 0,C 180,E1 -989.153,E2 -989.153} C_VEL
LIN {X 0,Y 594.387,Z 642.406,A -85,B 0,C 180,E1 -990.339,E2 -990.339} C_VEL
LIN {X 0,Y 594.459,Z 632.223,A -85,B 0,C 180,E1 -991.524,E2 -991.524} C_VEL
LIN {X 0,Y 594.528,Z 621.861,A -85,B 0,C 180,E1 -992.541,E2 -992.541} C_VEL
LIN {X 0,Y 594.602,Z 609.52,A -85,B 0,C 180,E1 -993.558,E2 -993.558} C_VEL
LIN {X 0,Y 594.726,Z 597.173,A -85,B 0,C 180,E1 -994.405,E2 -994.405} C_VEL
LIN {X 0,Y 594.788,Z 583.728,A -85,B 0,C 180,E1 -995.169,E2 -995.169} C_VEL
LIN {X 0,Y 594.906,Z 569.814,A -85,B 0,C 180,E1 -995.806,E2 -995.806} C_VEL
LIN {X 0,Y 595.002,Z 555.237,A -85,B 0,C 180,E1 -996.324,E2 -996.324} C_VEL
LIN {X 0,Y 595.062,Z 540.778,A -85,B 0,C 180,E1 -996.703,E2 -996.703} C_VEL
LIN {X 0,Y 595.105,Z 525.088,A -85,B 0,C 180,E1 -996.967,E2 -996.967} C_VEL
LIN {X 0,Y 595.219,Z 370.867,A -85,B 0,C 180,E1 -998.879,E2 -998.879} C_VEL
LIN {X 0,Y 594.643,Z 367.898,A -85,B 0,C 180,E1 -998.945,E2 -998.945} C_VEL
LIN {X 0,Y 594.753,Z 346.921,A -85,B 0,C 180,E1 -1001.762,E2 -1001.762} C_VEL
LIN {X 0,Y 594.68,Z 341.839,A -85,B 0,C 180,E1 -1002.456,E2 -1002.456} C_VEL
LIN {X 0,Y 594.343,Z 340.076,A -85,B 0,C 180,E1 -1002.723,E2 -1002.723} C_VEL
LIN {X 0,Y 594.348,Z 340.074,A -85,B 0,C 180,E1 -1005.079,E2 -1005.079} C_VEL
LIN {X 0,Y 594.374,Z 340.072,A -85,B 0,C 180,E1 -1007.194,E2 -1007.194} C_VEL
LIN {X 0,Y 594.365,Z 340.07,A -85,B 0,C 180,E1 -1010.054,E2 -1010.054} C_VEL
LIN {X 0,Y 594.354,Z 340.071,A -85,B 0,C 180,E1 -1012.968,E2 -1012.968} C_VEL
LIN {X 0,Y 594.371,Z 340.071,A -85,B 0,C 180,E1 -1015.193,E2 -1015.193} C_VEL
LIN {X 0,Y 594.351,Z 340.08,A -85,B 0,C 180,E1 -1017.519,E2 -1017.519} C_VEL
LIN {X 0,Y 594.373,Z 340.067,A -85,B 0,C 180,E1 -1020.325,E2 -1020.325} C_VEL
LIN {X 0,Y 594.378,Z 340.067,A -85,B 0,C 180,E1 -1022.95,E2 -1022.95} C_VEL
LIN {X 0,Y 594.329,Z 340.08,A -85,B 0,C 180,E1 -1025.411,E2 -1025.411} C_VEL
LIN {X 0,Y 594.372,Z 340.07,A -85,B 0,C 180,E1 -1027.942,E2 -1027.942} C_VEL
LIN {X 0,Y 594.364,Z 340.067,A -85,B 0,C 180,E1 -1030.82,E2 -1030.82} C_VEL
LIN {X 0,Y 594.346,Z 340.076,A -85,B 0,C 180,E1 -1033.302,E2 -1033.302} C_VEL
LIN {X 0,Y 594.347,Z 340.07,A -85,B 0,C 180,E1 -1036.163,E2 -1036.163} C_VEL
LIN {X 0,Y 594.368,Z 340.067,A -85,B 0,C 180,E1 -1038.534,E2 -1038.534} C_VEL
LIN {X 0,Y 594.369,Z 340.072,A -85,B 0,C 180,E1 -1041.298,E2 -1041.298} C_VEL
LIN {X 0,Y 594.35,Z 340.076,A -85,B 0,C 180,E1 -1043.755,E2 -1043.755} C_VEL
LIN {X 0,Y 594.365,Z 340.068,A -85,B 0,C 180,E1 -1046.237,E2 -1046.237} C_VEL
LIN {X 0,Y 594.363,Z 340.067,A -85,B 0,C 180,E1 -1048.649,E2 -1048.649} C_VEL
LIN {X 0,Y 594.38,Z 340.067,A -85,B 0,C 180,E1 -1051.043,E2 -1051.043} C_VEL
LIN {X 0,Y 594.36,Z 340.068,A -85,B 0,C 180,E1 -1054.055,E2 -1054.055} C_VEL
LIN {X 0,Y 594.372,Z 340.066,A -85,B 0,C 180,E1 -1056.295,E2 -1056.295} C_VEL
LIN {X 0,Y 594.399,Z 340.067,A -85,B 0,C 180,E1 -1059.224,E2 -1059.224} C_VEL
LIN {X 0,Y 594.342,Z 340.072,A -85,B 0,C 180,E1 -1062.094,E2 -1062.094} C_VEL
LIN {X 0,Y 594.353,Z 340.07,A -85,B 0,C 180,E1 -1064.218,E2 -1064.218} C_VEL
LIN {X 0,Y 594.369,Z 340.067,A -85,B 0,C 180,E1 -1066.32,E2 -1066.32} C_VEL
LIN {X 0,Y 594.35,Z 340.071,A -85,B 0,C 180,E1 -1069.094,E2 -1069.094} C_VEL
LIN {X 0,Y 594.382,Z 340.071,A -85,B 0,C 180,E1 -1071.843,E2 -1071.843} C_VEL
LIN {X 0,Y 594.365,Z 340.066,A -85,B 0,C 180,E1 -1074.572,E2 -1074.572} C_VEL
LIN {X 0,Y 594.393,Z 340.069,A -85,B 0,C 180,E1 -1077.289,E2 -1077.289} C_VEL
LIN {X 0,Y 594.414,Z 340.064,A -85,B 0,C 180,E1 -1080,E2 -1080} C_VEL
LIN {X 0,Y 594.378,Z 340.065,A -85,B 0,C 180,E1 -1082.711,E2 -1082.711} C_VEL
LIN {X 0,Y 594.377,Z 340.073,A -85,B 0,C 180,E1 -1085.428,E2 -1085.428} C_VEL
LIN {X 0,Y 594.381,Z 340.067,A -85,B 0,C 180,E1 -1088.157,E2 -1088.157} C_VEL
LIN {X 0,Y 594.37,Z 340.069,A -85,B 0,C 180,E1 -1091.062,E2 -1091.062} C_VEL
LIN {X 0,Y 594.373,Z 340.075,A -85,B 0,C 180,E1 -1093.679,E2 -1093.679} C_VEL
LIN {X 0,Y 594.336,Z 340.07,A -85,B 0,C 180,E1 -1096.699,E2 -1096.699} C_VEL
LIN {X 0,Y 594.359,Z 340.073,A -85,B 0,C 180,E1 -1099.334,E2 -1099.334} C_VEL
LIN {X 0,Y 594.353,Z 340.077,A -85,B 0,C 180,E1 -1101.504,E2 -1101.504} C_VEL
LIN {X 0,Y 594.368,Z 340.067,A -85,B 0,C 180,E1 -1104.447,E2 -1104.447} C_VEL
LIN {X 0,Y 594.356,Z 340.068,A -85,B 0,C 180,E1 -1106.701,E2 -1106.701} C_VEL
LIN {X 0,Y 594.371,Z 340.068,A -85,B 0,C 180,E1 -1108.999,E2 -1108.999} C_VEL
LIN {X 0,Y 594.372,Z 340.077,A -85,B 0,C 180,E1 -1111.641,E2 -1111.641} C_VEL
LIN {X 0,Y 594.36,Z 340.068,A -85,B 0,C 180,E1 -1114.581,E2 -1114.581} C_VEL
LIN {X 0,Y 594.363,Z 340.078,A -85,B 0,C 180,E1 -1117.605,E2 -1117.605} C_VEL
LIN {X 0,Y 594.353,Z 340.068,A -85,B 0,C 180,E1 -1120.568,E2 -1120.568} C_VEL
LIN {X 0,Y 594.341,Z 340.075,A -85,B 0,C 180,E1 -1123.302,E2 -1123.302} C_VEL
LIN {X 0,Y 594.343,Z 340.073,A -85,B 0,C 180,E1 -1126.163,E2 -1126.163} C_VEL
LIN {X 0,Y 594.364,Z 340.068,A -85,B 0,C 180,E1 -1128.534,E2 -1128.534} C_VEL
LIN {X 0,Y 594.365,Z 340.072,A -85,B 0,C 180,E1 -1131.298,E2 -1131.298} C_VEL
LIN {X 0,Y 594.346,Z 340.079,A -85,B 0,C 180,E1 -1133.755,E2 -1133.755} C_VEL
LIN {X 0,Y 594.361,Z 340.07,A -85,B 0,C 180,E1 -1136.237,E2 -1136.237} C_VEL
LIN {X 0,Y 594.359,Z 340.068,A -85,B 0,C 180,E1 -1138.649,E2 -1138.649} C_VEL
LIN {X 0,Y 594.375,Z 340.068,A -85,B 0,C 180,E1 -1141.044,E2 -1141.044} C_VEL
LIN {X 0,Y 594.363,Z 340.075,A -85,B 0,C 180,E1 -1144.196,E2 -1144.196} C_VEL
LIN {X 0,Y 595.008,Z 343.461,A -85,B 0,C 180,E1 -1144.648,E2 -1144.648} C_VEL
LIN {X 0,Y 594.922,Z 363.841,A -85,B 0,C 180,E1 -1147.055,E2 -1147.055} C_VEL
LIN {X 0,Y 594.813,Z 385.789,A -85,B 0,C 180,E1 -1149.601,E2 -1149.601} C_VEL
LIN {X 0,Y 594.701,Z 398.859,A -85,B 0,C 180,E1 -1151.095,E2 -1151.095} C_VEL
LIN {X 0,Y 595.318,Z 402.422,A -85,B 0,C 180,E1 -1151.163,E2 -1151.163} C_VEL
LIN {X 0,Y 595.081,Z 565.388,A -85,B 0,C 180,E1 -1153.199,E2 -1153.199} C_VEL
LIN {X 0,Y 595.014,Z 580.706,A -85,B 0,C 180,E1 -1153.532,E2 -1153.532} C_VEL
LIN {X 0,Y 594.933,Z 596.044,A -85,B 0,C 180,E1 -1154.014,E2 -1154.014} C_VEL
LIN {X 0,Y 594.858,Z 609.76,A -85,B 0,C 180,E1 -1154.584,E2 -1154.584} C_VEL
LIN {X 0,Y 594.732,Z 623.234,A -85,B 0,C 180,E1 -1155.282,E2 -1155.282} C_VEL
LIN {X 0,Y 594.681,Z 635.791,A -85,B 0,C 180,E1 -1156.075,E2 -1156.075} C_VEL
LIN {X 0,Y 594.56,Z 648.285,A -85,B 0,C 180,E1 -1157.021,E2 -1157.021} C_VEL
LIN {X 0,Y 594.466,Z 659.747,A -85,B 0,C 180,E1 -1158.06,E2 -1158.06} C_VEL
LIN {X 0,Y 594.388,Z 669.389,A -85,B 0,C 180,E1 -1159.095,E2 -1159.095} C_VEL
LIN {X 0,Y 594.367,Z 678.855,A -85,B 0,C 180,E1 -1160.299,E2 -1160.299} C_VEL
LIN {X 0,Y 594.311,Z 686.73,A -85,B 0,C 180,E1 -1161.499,E2 -1161.499} C_VEL
LIN {X 0,Y 594.291,Z 694.088,A -85,B 0,C 180,E1 -1162.867,E2 -1162.867} C_VEL
LIN {X 0,Y 594.298,Z 699.924,A -85,B 0,C 180,E1 -1164.231,E2 -1164.231} C_VEL
LIN {X 0,Y 594.232,Z 703.383,A -85,B 0,C 180,E1 -1165.251,E2 -1165.251} C_VEL
LIN {X 0,Y 594.257,Z 706.887,A -85,B 0,C 180,E1 -1166.61,E2 -1166.61} C_VEL
LIN {X 0,Y 594.241,Z 709.193,A -85,B 0,C 180,E1 -1167.967,E2 -1167.967} C_VEL
LIN {X 0,Y 594.235,Z 710.35,A -85,B 0,C 180,E1 -1169.322,E2 -1169.322} C_VEL
LIN {X 0,Y 594.235,Z 710.35,A -85,B 0,C 180,E1 -1170.678,E2 -1170.678} C_VEL
LIN {X 0,Y 594.241,Z 709.192,A -85,B 0,C 180,E1 -1172.033,E2 -1172.033} C_VEL
LIN {X 0,Y 594.257,Z 706.886,A -85,B 0,C 180,E1 -1173.39,E2 -1173.39} C_VEL
LIN {X 0,Y 594.232,Z 703.384,A -85,B 0,C 180,E1 -1174.749,E2 -1174.749} C_VEL
LIN {X 0,Y 594.278,Z 698.608,A -85,B 0,C 180,E1 -1176.11,E2 -1176.11} C_VEL
LIN {X 0,Y 594.287,Z 692.425,A -85,B 0,C 180,E1 -1177.475,E2 -1177.475} C_VEL
LIN {X 0,Y 594.33,Z 684.652,A -85,B 0,C 180,E1 -1178.843,E2 -1178.843} C_VEL
LIN {X 0,Y 594.388,Z 676.37,A -85,B 0,C 180,E1 -1180.044,E2 -1180.044} C_VEL
LIN {X 0,Y 594.433,Z 666.559,A -85,B 0,C 180,E1 -1181.231,E2 -1181.231} C_VEL
LIN {X 0,Y 594.531,Z 656.191,A -85,B 0,C 180,E1 -1182.285,E2 -1182.285} C_VEL
LIN {X 0,Y 594.581,Z 644.016,A -85,B 0,C 180,E1 -1183.326,E2 -1183.326} C_VEL
LIN {X 0,Y 594.694,Z 632.074,A -85,B 0,C 180,E1 -1184.178,E2 -1184.178} C_VEL
LIN {X 0,Y 594.75,Z 618.524,A -85,B 0,C 180,E1 -1184.981,E2 -1184.981} C_VEL
LIN {X 0,Y 594.903,Z 603.839,A -85,B 0,C 180,E1 -1185.678,E2 -1185.678} C_VEL
LIN {X 0,Y 594.966,Z 589.616,A -85,B 0,C 180,E1 -1186.205,E2 -1186.205} C_VEL
LIN {X 0,Y 595.043,Z 575.131,A -85,B 0,C 180,E1 -1186.603,E2 -1186.603} C_VEL
LIN {X 0,Y 595.066,Z 559.746,A -85,B 0,C 180,E1 -1186.886,E2 -1186.886} C_VEL
LIN {X 0,Y 595.219,Z 401.517,A -85,B 0,C 180,E1 -1188.851,E2 -1188.851} C_VEL
LIN {X 0,Y 594.733,Z 398.771,A -85,B 0,C 180,E1 -1188.914,E2 -1188.914} C_VEL
LIN {X 0,Y 594.894,Z 373.248,A -85,B 0,C 180,E1 -1191.848,E2 -1191.848} C_VEL
LIN {X 0,Y 595.048,Z 349.985,A -85,B 0,C 180,E1 -1194.573,E2 -1194.573} C_VEL
LIN {X 0,Y 595.007,Z 343.462,A -85,B 0,C 180,E1 -1195.352,E2 -1195.352} C_VEL
LIN {X 0,Y 594.361,Z 340.076,A -85,B 0,C 180,E1 -1195.804,E2 -1195.804} C_VEL
LIN {X 0,Y 594.375,Z 340.068,A -85,B 0,C 180,E1 -1198.956,E2 -1198.956} C_VEL
LIN {X 0,Y 594.371,Z 340.068,A -85,B 0,C 180,E1 -1201.642,E2 -1201.642} C_VEL
LIN {X 0,Y 594.367,Z 340.074,A -85,B 0,C 180,E1 -1204.137,E2 -1204.137} C_VEL
LIN {X 0,Y 594.331,Z 340.072,A -85,B 0,C 180,E1 -1207.091,E2 -1207.091} C_VEL
LIN {X 0,Y 594.345,Z 340.071,A -85,B 0,C 180,E1 -1209.771,E2 -1209.771} C_VEL
LIN {X 0,Y 594.365,Z 340.077,A -85,B 0,C 180,E1 -1212.376,E2 -1212.376} C_VEL
LIN {X 0,Y 594.336,Z 340.071,A -85,B 0,C 180,E1 -1215.194,E2 -1215.194} C_VEL
LIN {X 0,Y 594.376,Z 340.073,A -85,B 0,C 180,E1 -1218.153,E2 -1218.153} C_VEL
LIN {X 0,Y 594.364,Z 340.067,A -85,B 0,C 180,E1 -1221.298,E2 -1221.298} C_VEL
LIN {X 0,Y 594.345,Z 340.07,A -85,B 0,C 180,E1 -1223.755,E2 -1223.755} C_VEL
LIN {X 0,Y 594.375,Z 340.073,A -85,B 0,C 180,E1 -1226.239,E2 -1226.239} C_VEL
LIN {X 0,Y 594.361,Z 340.072,A -85,B 0,C 180,E1 -1228.649,E2 -1228.649} C_VEL
LIN {X 0,Y 594.372,Z 340.067,A -85,B 0,C 180,E1 -1231.044,E2 -1231.044} C_VEL
LIN {X 0,Y 594.357,Z 340.068,A -85,B 0,C 180,E1 -1233.299,E2 -1233.299} C_VEL
LIN {X 0,Y 594.356,Z 340.068,A -85,B 0,C 180,E1 -1235.574,E2 -1235.574} C_VEL
LIN {X 0,Y 594.355,Z 340.078,A -85,B 0,C 180,E1 -1238.496,E2 -1238.496} C_VEL
LIN {X 0,Y 594.355,Z 340.068,A -85,B 0,C 180,E1 -1241.382,E2 -1241.382} C_VEL
LIN {X 0,Y 594.353,Z 340.075,A -85,B 0,C 180,E1 -1244.219,E2 -1244.219} C_VEL
LIN {X 0,Y 594.375,Z 340.075,A -85,B 0,C 180,E1 -1246.321,E2 -1246.321} C_VEL
LIN {X 0,Y 594.352,Z 340.07,A -85,B 0,C 180,E1 -1249.094,E2 -1249.094} C_VEL
LIN {X 0,Y 594.381,Z 340.066,A -85,B 0,C 180,E1 -1251.843,E2 -1251.843} C_VEL
LIN {X 0,Y 594.381,Z 340.073,A -85,B 0,C 180,E1 -1254.572,E2 -1254.572} C_VEL
LIN {X 0,Y 594.381,Z 340.065,A -85,B 0,C 180,E1 -1257.289,E2 -1257.289} C_VEL
LIN {X 0,Y 594.414,Z 340.064,A -85,B 0,C 180,E1 -1260,E2 -1260} C_VEL
LIN {X 0,Y 594.398,Z 340.069,A -85,B 0,C 180,E1 -1262.711,E2 -1262.711} C_VEL
LIN {X 0,Y 594.368,Z 340.067,A -85,B 0,C 180,E1 -1265.428,E2 -1265.428} C_VEL
LIN {X 0,Y 594.383,Z 340.069,A -85,B 0,C 180,E1 -1268.157,E2 -1268.157} C_VEL
LIN {X 0,Y 594.372,Z 340.068,A -85,B 0,C 180,E1 -1271.064,E2 -1271.064} C_VEL
LIN {X 0,Y 594.371,Z 340.067,A -85,B 0,C 180,E1 -1273.68,E2 -1273.68} C_VEL
LIN {X 0,Y 594.349,Z 340.069,A -85,B 0,C 180,E1 -1275.324,E2 -1275.324} C_VEL
LIN {X 0,Y 593.674,Z 340.156,A -85,B 0,C 180,E1 -1275.89,E2 -1275.89} C_VEL
LIN {X 0,Y 590.81,Z 340.515,A -85,B 0,C 180,E1 -1276.807,E2 -1276.807} C_VEL
LIN {X 0,Y 588.403,Z 340.816,A -85,B 0,C 180,E1 -1277.546,E2 -1277.546} C_VEL
LIN {X 0,Y 587.383,Z 340.941,A -85,B 0,C 180,E1 -1278.116,E2 -1278.116} C_VEL
LIN {X 0,Y 587.306,Z 340.949,A -85,B 0,C 180,E1 -1278.309,E2 -1278.309} C_VEL
LIN {X 0,Y 587.335,Z 340.945,A -85,B 0,C 180,E1 -1281.038,E2 -1281.038} C_VEL
LIN {X 0,Y 587.313,Z 340.946,A -85,B 0,C 180,E1 -1283.26,E2 -1283.26} C_VEL
LIN {X 0,Y 587.319,Z 340.943,A -85,B 0,C 180,E1 -1285.518,E2 -1285.518} C_VEL
LIN {X 0,Y 587.322,Z 340.954,A -85,B 0,C 180,E1 -1288.598,E2 -1288.598} C_VEL
LIN {X 0,Y 587.326,Z 340.946,A -85,B 0,C 180,E1 -1290.967,E2 -1290.967} C_VEL
LIN {X 0,Y 587.33,Z 340.944,A -85,B 0,C 180,E1 -1293.397,E2 -1293.397} C_VEL
LIN {X 0,Y 587.285,Z 340.949,A -85,B 0,C 180,E1 -1295.901,E2 -1295.901} C_VEL
LIN {X 0,Y 587.32,Z 340.955,A -85,B 0,C 180,E1 -1298.481,E2 -1298.481} C_VEL
LIN {X 0,Y 587.314,Z 340.947,A -85,B 0,C 180,E1 -1301.159,E2 -1301.159} C_VEL
LIN {X 0,Y 587.307,Z 340.95,A -85,B 0,C 180,E1 -1304.111,E2 -1304.111} C_VEL
LIN {X 0,Y 587.297,Z 340.951,A -85,B 0,C 180,E1 -1306.992,E2 -1306.992} C_VEL
LIN {X 0,Y 587.309,Z 340.947,A -85,B 0,C 180,E1 -1309.745,E2 -1309.745} C_VEL
LIN {X 0,Y 587.344,Z 340.95,A -85,B 0,C 180,E1 -1312.392,E2 -1312.392} C_VEL
LIN {X 0,Y 587.356,Z 340.943,A -85,B 0,C 180,E1 -1315.78,E2 -1315.78} C_VEL
LIN {X 0,Y 587.37,Z 341.154,A -85,B 0,C 180,E1 -1317.245,E2 -1317.245} C_VEL
LIN {X 0,Y 587.865,Z 345.158,A -85,B 0,C 180,E1 -1317.818,E2 -1317.818} C_VEL
LIN {X 0,Y 587.705,Z 364.426,A -85,B 0,C 180,E1 -1320.443,E2 -1320.443} C_VEL
LIN {X 0,Y 587.728,Z 368.259,A -85,B 0,C 180,E1 -1320.928,E2 -1320.928} C_VEL
LIN {X 0,Y 588.529,Z 372.004,A -85,B 0,C 180,E1 -1321.003,E2 -1321.003} C_VEL
LIN {X 0,Y 588.304,Z 532.247,A -85,B 0,C 180,E1 -1323.026,E2 -1323.026} C_VEL
LIN {X 0,Y 588.226,Z 546.818,A -85,B 0,C 180,E1 -1323.334,E2 -1323.334} C_VEL
LIN {X 0,Y 588.078,Z 561.687,A -85,B 0,C 180,E1 -1323.785,E2 -1323.785} C_VEL
LIN {X 0,Y 587.995,Z 576.153,A -85,B 0,C 180,E1 -1324.372,E2 -1324.372} C_VEL
LIN {X 0,Y 587.817,Z 589.896,A -85,B 0,C 180,E1 -1325.074,E2 -1325.074} C_VEL
LIN {X 0,Y 587.713,Z 603.343,A -85,B 0,C 180,E1 -1325.92,E2 -1325.92} C_VEL
LIN {X 0,Y 587.62,Z 615.653,A -85,B 0,C 180,E1 -1326.857,E2 -1326.857} C_VEL
LIN {X 0,Y 587.498,Z 626.755,A -85,B 0,C 180,E1 -1327.863,E2 -1327.863} C_VEL
LIN {X 0,Y 587.374,Z 637.014,A -85,B 0,C 180,E1 -1328.964,E2 -1328.964} C_VEL
LIN {X 0,Y 587.286,Z 646.959,A -85,B 0,C 180,E1 -1330.241,E2 -1330.241} C_VEL
LIN {X 0,Y 587.25,Z 655.128,A -85,B 0,C 180,E1 -1331.51,E2 -1331.51} C_VEL
LIN {X 0,Y 587.24,Z 660.986,A -85,B 0,C 180,E1 -1332.591,E2 -1332.591} C_VEL
LIN {X 0,Y 587.197,Z 667.257,A -85,B 0,C 180,E1 -1334.021,E2 -1334.021} C_VEL
LIN {X 0,Y 587.161,Z 672.01,A -85,B 0,C 180,E1 -1335.442,E2 -1335.442} C_VEL
LIN {X 0,Y 587.144,Z 675.388,A -85,B 0,C 180,E1 -1336.854,E2 -1336.854} C_VEL
LIN {X 0,Y 587.155,Z 677.502,A -85,B 0,C 180,E1 -1338.259,E2 -1338.259} C_VEL
LIN {X 0,Y 587.137,Z 678.418,A -85,B 0,C 180,E1 -1339.657,E2 -1339.657} C_VEL
LIN {X 0,Y 587.122,Z 678.164,A -85,B 0,C 180,E1 -1341.048,E2 -1341.048} C_VEL
LIN {X 0,Y 587.128,Z 676.758,A -85,B 0,C 180,E1 -1342.434,E2 -1342.434} C_VEL
LIN {X 0,Y 587.146,Z 674.172,A -85,B 0,C 180,E1 -1343.816,E2 -1343.816} C_VEL
LIN {X 0,Y 587.139,Z 670.33,A -85,B 0,C 180,E1 -1345.194,E2 -1345.194} C_VEL
LIN {X 0,Y 587.197,Z 665.203,A -85,B 0,C 180,E1 -1346.569,E2 -1346.569} C_VEL
LIN {X 0,Y 587.21,Z 658.685,A -85,B 0,C 180,E1 -1347.942,E2 -1347.942} C_VEL
LIN {X 0,Y 587.303,Z 650.59,A -85,B 0,C 180,E1 -1349.314,E2 -1349.314} C_VEL
LIN {X 0,Y 587.337,Z 642.012,A -85,B 0,C 180,E1 -1350.514,E2 -1350.514} C_VEL
LIN {X 0,Y 587.462,Z 631.749,A -85,B 0,C 180,E1 -1351.714,E2 -1351.714} C_VEL
LIN {X 0,Y 587.513,Z 621.308,A -85,B 0,C 180,E1 -1352.743,E2 -1352.743} C_VEL
LIN {X 0,Y 587.666,Z 608.848,A -85,B 0,C 180,E1 -1353.771,E2 -1353.771} C_VEL
LIN {X 0,Y 587.822,Z 596.357,A -85,B 0,C 180,E1 -1354.629,E2 -1354.629} C_VEL
LIN {X 0,Y 587.912,Z 582.718,A -85,B 0,C 180,E1 -1355.402,E2 -1355.402} C_VEL
LIN {X 0,Y 588.076,Z 568.51,A -85,B 0,C 180,E1 -1356.045,E2 -1356.045} C_VEL
LIN {X 0,Y 588.157,Z 553.801,A -85,B 0,C 180,E1 -1356.561,E2 -1356.561} C_VEL
LIN {X 0,Y 588.264,Z 538.991,A -85,B 0,C 180,E1 -1356.937,E2 -1356.937} C_VEL
LIN {X 0,Y 588.307,Z 523.503,A -85,B 0,C 180,E1 -1357.189,E2 -1357.189} C_VEL
LIN {X 0,Y 588.59,Z 372.309,A -85,B 0,C 180,E1 -1359.081,E2 -1359.081} C_VEL
LIN {X 0,Y 587.688,Z 367.865,A -85,B 0,C 180,E1 -1359.182,E2 -1359.182} C_VEL
LIN {X 0,Y 587.889,Z 346.574,A -85,B 0,C 180,E1 -1362.076,E2 -1362.076} C_VEL
LIN {X 0,Y 587.413,Z 341.553,A -85,B 0,C 180,E1 -1362.788,E2 -1362.788} C_VEL
LIN {X 0,Y 587.319,Z 340.952,A -85,B 0,C 180,E1 -1362.878,E2 -1362.878} C_VEL
LIN {X 0,Y 587.312,Z 340.954,A -85,B 0,C 180,E1 -1365.264,E2 -1365.264} C_VEL
LIN {X 0,Y 587.31,Z 340.956,A -85,B 0,C 180,E1 -1367.407,E2 -1367.407} C_VEL
LIN {X 0,Y 587.31,Z 340.956,A -85,B 0,C 180,E1 -1369.576,E2 -1369.576} C_VEL
LIN {X 0,Y 587.315,Z 340.952,A -85,B 0,C 180,E1 -1371.775,E2 -1371.775} C_VEL
LIN {X 0,Y 587.317,Z 340.946,A -85,B 0,C 180,E1 -1374.76,E2 -1374.76} C_VEL
LIN {X 0,Y 587.307,Z 340.955,A -85,B 0,C 180,E1 -1377.683,E2 -1377.683} C_VEL
LIN {X 0,Y 587.32,Z 340.946,A -85,B 0,C 180,E1 -1380.171,E2 -1380.171} C_VEL
LIN {X 0,Y 587.333,Z 340.942,A -85,B 0,C 180,E1 -1382.58,E2 -1382.58} C_VEL
LIN {X 0,Y 587.307,Z 340.949,A -85,B 0,C 180,E1 -1385.057,E2 -1385.057} C_VEL
LIN {X 0,Y 587.324,Z 340.95,A -85,B 0,C 180,E1 -1387.836,E2 -1387.836} C_VEL
LIN {X 0,Y 587.308,Z 340.946,A -85,B 0,C 180,E1 -1390.255,E2 -1390.255} C_VEL
LIN {X 0,Y 587.29,Z 340.952,A -85,B 0,C 180,E1 -1393.115,E2 -1393.115} C_VEL
LIN {X 0,Y 587.303,Z 340.949,A -85,B 0,C 180,E1 -1396.047,E2 -1396.047} C_VEL
LIN {X 0,Y 587.312,Z 340.947,A -85,B 0,C 180,E1 -1398.84,E2 -1398.84} C_VEL
LIN {X 0,Y 587.318,Z 340.955,A -85,B 0,C 180,E1 -1401.519,E2 -1401.519} C_VEL
LIN {X 0,Y 587.282,Z 340.952,A -85,B 0,C 180,E1 -1404.099,E2 -1404.099} C_VEL
LIN {X 0,Y 587.33,Z 340.943,A -85,B 0,C 180,E1 -1406.602,E2 -1406.602} C_VEL
LIN {X 0,Y 587.322,Z 340.947,A -85,B 0,C 180,E1 -1409.032,E2 -1409.032} C_VEL
LIN {X 0,Y 587.321,Z 340.952,A -85,B 0,C 180,E1 -1411.402,E2 -1411.402} C_VEL
LIN {X 0,Y 587.307,Z 340.943,A -85,B 0,C 180,E1 -1414.482,E2 -1414.482} C_VEL
LIN {X 0,Y 587.312,Z 340.948,A -85,B 0,C 180,E1 -1417.134,E2 -1417.134} C_VEL
LIN {X 0,Y 587.323,Z 340.953,A -85,B 0,C 180,E1 -1419.695,E2 -1419.695} C_VEL
LIN {X 0,Y 587.297,Z 340.952,A -85,B 0,C 180,E1 -1421.872,E2 -1421.872} C_VEL
LIN {X 0,Y 587.31,Z 340.949,A -85,B 0,C 180,E1 -1424.024,E2 -1424.024} C_VEL
LIN {X 0,Y 587.352,Z 340.942,A -85,B 0,C 180,E1 -1426.154,E2 -1426.154} C_VEL
LIN {X 0,Y 587.341,Z 340.942,A -85,B 0,C 180,E1 -1428.962,E2 -1428.962} C_VEL
LIN {X 0,Y 587.341,Z 340.95,A -85,B 0,C 180,E1 -1431.744,E2 -1431.744} C_VEL
LIN {X 0,Y 587.334,Z 340.942,A -85,B 0,C 180,E1 -1434.506,E2 -1434.506} C_VEL
LIN {X 0,Y 587.358,Z 340.944,A -85,B 0,C 180,E1 -1437.256,E2 -1437.256} C_VEL
LIN {X 0,Y 587.383,Z 340.94,A -85,B 0,C 180,E1 -1440,E2 -1440} C_VEL
LIN {X 0,Y 587.348,Z 340.941,A -85,B 0,C 180,E1 -1442.743,E2 -1442.743} C_VEL
LIN {X 0,Y 587.344,Z 340.95,A -85,B 0,C 180,E1 -1445.493,E2 -1445.493} C_VEL
LIN {X 0,Y 587.339,Z 340.943,A -85,B 0,C 180,E1 -1448.255,E2 -1448.255} C_VEL
LIN {X 0,Y 587.333,Z 340.946,A -85,B 0,C 180,E1 -1451.124,E2 -1451.124} C_VEL
LIN {X 0,Y 587.342,Z 340.943,A -85,B 0,C 180,E1 -1454.25,E2 -1454.25} C_VEL
LIN {X 0,Y 587.288,Z 340.949,A -85,B 0,C 180,E1 -1456.793,E2 -1456.793} C_VEL
LIN {X 0,Y 587.305,Z 340.956,A -85,B 0,C 180,E1 -1459.576,E2 -1459.576} C_VEL
LIN {X 0,Y 587.309,Z 340.953,A -85,B 0,C 180,E1 -1461.775,E2 -1461.775} C_VEL
LIN {X 0,Y 587.313,Z 340.946,A -85,B 0,C 180,E1 -1464.76,E2 -1464.76} C_VEL
LIN {X 0,Y 587.302,Z 340.957,A -85,B 0,C 180,E1 -1467.683,E2 -1467.683} C_VEL
LIN {X 0,Y 587.316,Z 340.947,A -85,B 0,C 180,E1 -1470.171,E2 -1470.171} C_VEL
LIN {X 0,Y 587.329,Z 340.943,A -85,B 0,C 180,E1 -1472.579,E2 -1472.579} C_VEL
LIN {X 0,Y 587.302,Z 340.949,A -85,B 0,C 180,E1 -1475.057,E2 -1475.057} C_VEL
LIN {X 0,Y 587.32,Z 340.951,A -85,B 0,C 180,E1 -1477.836,E2 -1477.836} C_VEL
LIN {X 0,Y 587.303,Z 340.948,A -85,B 0,C 180,E1 -1480.255,E2 -1480.255} C_VEL
LIN {X 0,Y 587.285,Z 340.952,A -85,B 0,C 180,E1 -1483.115,E2 -1483.115} C_VEL
LIN {X 0,Y 587.298,Z 340.952,A -85,B 0,C 180,E1 -1486.047,E2 -1486.047} C_VEL
LIN {X 0,Y 587.307,Z 340.947,A -85,B 0,C 180,E1 -1488.84,E2 -1488.84} C_VEL
LIN {X 0,Y 587.314,Z 340.955,A -85,B 0,C 180,E1 -1491.519,E2 -1491.519} C_VEL
LIN {X 0,Y 587.278,Z 340.954,A -85,B 0,C 180,E1 -1494.099,E2 -1494.099} C_VEL
LIN {X 0,Y 587.325,Z 340.945,A -85,B 0,C 180,E1 -1496.603,E2 -1496.603} C_VEL
LIN {X 0,Y 587.331,Z 340.952,A -85,B 0,C 180,E1 -1499.491,E2 -1499.491} C_VEL
LIN {X 0,Y 587.302,Z 340.952,A -85,B 0,C 180,E1 -1502.18,E2 -1502.18} C_VEL
LIN {X 0,Y 587.347,Z 341.067,A -85,B 0,C 180,E1 -1504.003,E2 -1504.003} C_VEL
LIN {X 0,Y 588.195,Z 345.029,A -85,B 0,C 180,E1 -1504.523,E2 -1504.523} C_VEL
LIN {X 0,Y 588.107,Z 363.841,A -85,B 0,C 180,E1 -1506.774,E2 -1506.774} C_VEL
LIN {X 0,Y 587.896,Z 387.356,A -85,B 0,C 180,E1 -1509.533,E2 -1509.533} C_VEL
LIN {X 0,Y 587.815,Z 399.023,A -85,B 0,C 180,E1 -1510.871,E2 -1510.871} C_VEL
LIN {X 0,Y 588.594,Z 403.556,A -85,B 0,C 180,E1 -1510.954,E2 -1510.954} C_VEL
LIN {X 0,Y 588.299,Z 565.379,A -85,B 0,C 180,E1 -1513,E2 -1513} C_VEL
LIN {X 0,Y 588.208,Z 580.705,A -85,B 0,C 180,E1 -1513.336,E2 -1513.336} C_VEL
LIN {X 0,Y 588.071,Z 596.042,A -85,B 0,C 180,E1 -1513.823,E2 -1513.823} C_VEL
LIN {X 0,Y 587.989,Z 609.762,A -85,B 0,C 180,E1 -1514.399,E2 -1514.399} C_VEL
LIN {X 0,Y 587.828,Z 623.236,A -85,B 0,C 180,E1 -1515.105,E2 -1515.105} C_VEL
LIN {X 0,Y 587.741,Z 636.112,A -85,B 0,C 180,E1 -1515.929,E2 -1515.929} C_VEL
LIN {X 0,Y 587.582,Z 648.286,A -85,B 0,C 180,E1 -1516.864,E2 -1516.864} C_VEL
LIN {X 0,Y 587.454,Z 659.748,A -85,B 0,C 180,E1 -1517.915,E2 -1517.915} C_VEL
LIN {X 0,Y 587.348,Z 669.389,A -85,B 0,C 180,E1 -1518.962,E2 -1518.962} C_VEL
LIN {X 0,Y 587.305,Z 678.855,A -85,B 0,C 180,E1 -1520.182,E2 -1520.182} C_VEL
LIN {X 0,Y 587.264,Z 686.731,A -85,B 0,C 180,E1 -1521.397,E2 -1521.397} C_VEL
LIN {X 0,Y 587.215,Z 694.088,A -85,B 0,C 180,E1 -1522.781,E2 -1522.781} C_VEL
LIN {X 0,Y 587.226,Z 699.924,A -85,B 0,C 180,E1 -1524.161,E2 -1524.161} C_VEL
LIN {X 0,Y 587.136,Z 703.384,A -85,B 0,C 180,E1 -1525.194,E2 -1525.194} C_VEL
LIN {X 0,Y 587.18,Z 706.888,A -85,B 0,C 180,E1 -1526.569,E2 -1526.569} C_VEL
LIN {X 0,Y 587.14,Z 709.193,A -85,B 0,C 180,E1 -1527.942,E2 -1527.942} C_VEL
LIN {X 0,Y 587.135,Z 710.35,A -85,B 0,C 180,E1 -1529.314,E2 -1529.314} C_VEL
LIN {X 0,Y 587.135,Z 710.35,A -85,B 0,C 180,E1 -1530.686,E2 -1530.686} C_VEL
LIN {X 0,Y 587.139,Z 709.193,A -85,B 0,C 180,E1 -1532.058,E2 -1532.058} C_VEL
LIN {X 0,Y 587.18,Z 706.886,A -85,B 0,C 180,E1 -1533.431,E2 -1533.431} C_VEL
LIN {X 0,Y 587.136,Z 703.384,A -85,B 0,C 180,E1 -1534.806,E2 -1534.806} C_VEL
LIN {X 0,Y 587.179,Z 698.608,A -85,B 0,C 180,E1 -1536.184,E2 -1536.184} C_VEL
LIN {X 0,Y 587.23,Z 692.424,A -85,B 0,C 180,E1 -1537.565,E2 -1537.565} C_VEL
LIN {X 0,Y 587.265,Z 684.651,A -85,B 0,C 180,E1 -1538.95,E2 -1538.95} C_VEL
LIN {X 0,Y 587.352,Z 676.37,A -85,B 0,C 180,E1 -1540.165,E2 -1540.165} C_VEL
LIN {X 0,Y 587.399,Z 666.395,A -85,B 0,C 180,E1 -1541.386,E2 -1541.386} C_VEL
LIN {X 0,Y 587.522,Z 656.19,A -85,B 0,C 180,E1 -1542.434,E2 -1542.434} C_VEL
LIN {X 0,Y 587.629,Z 644.017,A -85,B 0,C 180,E1 -1543.487,E2 -1543.487} C_VEL
LIN {X 0,Y 587.774,Z 631.055,A -85,B 0,C 180,E1 -1544.416,E2 -1544.416} C_VEL
LIN {X 0,Y 587.887,Z 616.865,A -85,B 0,C 180,E1 -1545.248,E2 -1545.248} C_VEL
LIN {X 0,Y 588.049,Z 602.795,A -85,B 0,C 180,E1 -1545.91,E2 -1545.91} C_VEL
LIN {X 0,Y 588.166,Z 588.302,A -85,B 0,C 180,E1 -1546.442,E2 -1546.442} C_VEL
LIN {X 0,Y 588.266,Z 572.455,A -85,B 0,C 180,E1 -1546.863,E2 -1546.863} C_VEL
LIN {X 0,Y 588.335,Z 556.617,A -85,B 0,C 180,E1 -1547.129,E2 -1547.129} C_VEL
LIN {X 0,Y 588.506,Z 402.396,A -85,B 0,C 180,E1 -1549.063,E2 -1549.063} C_VEL
LIN {X 0,Y 587.806,Z 398.742,A -85,B 0,C 180,E1 -1549.148,E2 -1549.148} C_VEL
LIN {X 0,Y 588.033,Z 373.248,A -85,B 0,C 180,E1 -1552.116,E2 -1552.116} C_VEL
LIN {X 0,Y 588.244,Z 349.891,A -85,B 0,C 180,E1 -1554.888,E2 -1554.888} C_VEL
LIN {X 0,Y 588.194,Z 345.03,A -85,B 0,C 180,E1 -1555.477,E2 -1555.477} C_VEL
LIN {X 0,Y 587.328,Z 340.953,A -85,B 0,C 180,E1 -1556.023,E2 -1556.023} C_VEL
LIN {X 0,Y 587.342,Z 340.943,A -85,B 0,C 180,E1 -1559.132,E2 -1559.132} C_VEL
LIN {X 0,Y 587.339,Z 340.946,A -85,B 0,C 180,E1 -1561.835,E2 -1561.835} C_VEL
LIN {X 0,Y 587.333,Z 340.954,A -85,B 0,C 180,E1 -1564.346,E2 -1564.346} C_VEL
LIN {X 0,Y 587.318,Z 340.946,A -85,B 0,C 180,E1 -1567.61,E2 -1567.61} C_VEL
LIN {X 0,Y 587.305,Z 340.955,A -85,B 0,C 180,E1 -1570.255,E2 -1570.255} C_VEL
LIN {X 0,Y 587.301,Z 340.949,A -85,B 0,C 180,E1 -1573.008,E2 -1573.008} C_VEL
LIN {X 0,Y 587.299,Z 340.952,A -85,B 0,C 180,E1 -1576.047,E2 -1576.047} C_VEL
LIN {X 0,Y 587.309,Z 340.949,A -85,B 0,C 180,E1 -1578.928,E2 -1578.928} C_VEL
LIN {X 0,Y 587.312,Z 340.946,A -85,B 0,C 180,E1 -1581.519,E2 -1581.519} C_VEL
LIN {X 0,Y 587.28,Z 340.954,A -85,B 0,C 180,E1 -1584.099,E2 -1584.099} C_VEL
LIN {X 0,Y 587.331,Z 340.95,A -85,B 0,C 180,E1 -1586.603,E2 -1586.603} C_VEL
LIN {X 0,Y 587.318,Z 340.944,A -85,B 0,C 180,E1 -1589.033,E2 -1589.033} C_VEL
LIN {X 0,Y 587.308,Z 340.946,A -85,B 0,C 180,E1 -1591.402,E2 -1591.402} C_VEL
LIN {X 0,Y 587.31,Z 340.947,A -85,B 0,C 180,E1 -1593.829,E2 -1593.829} C_VEL
LIN {X 0,Y 587.304,Z 340.95,A -85,B 0,C 180,E1 -1595.992,E2 -1595.992} C_VEL
LIN {X 0,Y 587.333,Z 340.945,A -85,B 0,C 180,E1 -1598.963,E2 -1598.963} C_VEL
LIN {X 0,Y 587.288,Z 340.951,A -85,B 0,C 180,E1 -1601.872,E2 -1601.872} C_VEL
LIN {X 0,Y 587.302,Z 340.951,A -85,B 0,C 180,E1 -1604.024,E2 -1604.024} C_VEL
LIN {X 0,Y 587.355,Z 340.946,A -85,B 0,C 180,E1 -1606.154,E2 -1606.154} C_VEL
LIN {X 0,Y 587.339,Z 340.945,A -85,B 0,C 180,E1 -1608.963,E2 -1608.963} C_VEL
LIN {X 0,Y 587.339,Z 340.943,A -85,B 0,C 180,E1 -1611.745,E2 -1611.745} C_VEL
LIN {X 0,Y 587.347,Z 340.951,A -85,B 0,C 180,E1 -1614.507,E2 -1614.507} C_VEL
LIN {X 0,Y 587.35,Z 340.941,A -85,B 0,C 180,E1 -1617.257,E2 -1617.257} C_VEL
LIN {X 0,Y 587.383,Z 340.939,A -85,B 0,C 180,E1 -1620,E2 -1620} C_VEL
LIN {X 0,Y 587.363,Z 340.944,A -85,B 0,C 180,E1 -1622.744,E2 -1622.744} C_VEL
LIN {X 0,Y 587.337,Z 340.943,A -85,B 0,C 180,E1 -1625.493,E2 -1625.493} C_VEL
LIN {X 0,Y 587.342,Z 340.948,A -85,B 0,C 180,E1 -1628.256,E2 -1628.256} C_VEL
LIN {X 0,Y 587.352,Z 340.942,A -85,B 0,C 180,E1 -1631.134,E2 -1631.134} C_VEL
LIN {X 0,Y 587.368,Z 340.945,A -85,B 0,C 180,E1 -1634.26,E2 -1634.26} C_VEL
LIN {X 0,Y 587.311,Z 340.946,A -85,B 0,C 180,E1 -1637.408,E2 -1637.408} C_VEL
LIN {X 0,Y 587.306,Z 340.949,A -85,B 0,C 180,E1 -1638.309,E2 -1638.309} C_VEL
LIN {X 0,Y 586.665,Z 341.028,A -85,B 0,C 180,E1 -1638.881,E2 -1638.881} C_VEL
LIN {X 0,Y 583.845,Z 341.378,A -85,B 0,C 180,E1 -1639.809,E2 -1639.809} C_VEL
LIN {X 0,Y 581.436,Z 341.686,A -85,B 0,C 180,E1 -1640.556,E2 -1640.556} C_VEL
LIN {X 0,Y 580.381,Z 341.811,A -85,B 0,C 180,E1 -1641.133,E2 -1641.133} C_VEL
LIN {X 0,Y 580.285,Z 341.821,A -85,B 0,C 180,E1 -1641.328,E2 -1641.328} C_VEL
LIN {X 0,Y 580.299,Z 341.827,A -85,B 0,C 180,E1 -1644.317,E2 -1644.317} C_VEL
LIN {X 0,Y 580.249,Z 341.826,A -85,B 0,C 180,E1 -1647.404,E2 -1647.404} C_VEL
LIN {X 0,Y 580.286,Z 341.821,A -85,B 0,C 180,E1 -1649.773,E2 -1649.773} C_VEL
LIN {X 0,Y 580.3,Z 341.823,A -85,B 0,C 180,E1 -1652.201,E2 -1652.201} C_VEL
LIN {X 0,Y 580.283,Z 341.827,A -85,B 0,C 180,E1 -1654.697,E2 -1654.697} C_VEL
LIN {X 0,Y 580.278,Z 341.823,A -85,B 0,C 180,E1 -1657.271,E2 -1657.271} C_VEL
LIN {X 0,Y 580.291,Z 341.826,A -85,B 0,C 180,E1 -1660.27,E2 -1660.27} C_VEL
LIN {X 0,Y 580.274,Z 341.831,A -85,B 0,C 180,E1 -1662.707,E2 -1662.707} C_VEL
LIN {X 0,Y 580.259,Z 341.824,A -85,B 0,C 180,E1 -1665.611,E2 -1665.611} C_VEL
LIN {X 0,Y 580.277,Z 341.831,A -85,B 0,C 180,E1 -1668.67,E2 -1668.67} C_VEL
LIN {X 0,Y 580.272,Z 341.827,A -85,B 0,C 180,E1 -1670.964,E2 -1670.964} C_VEL
LIN {X 0,Y 580.251,Z 341.826,A -85,B 0,C 180,E1 -1673.595,E2 -1673.595} C_VEL
LIN {X 0,Y 580.315,Z 341.824,A -85,B 0,C 180,E1 -1676.145,E2 -1676.145} C_VEL
LIN {X 0,Y 580.326,Z 341.883,A -85,B 0,C 180,E1 -1677.055,E2 -1677.055} C_VEL
LIN {X 0,Y 580.945,Z 347.311,A -85,B 0,C 180,E1 -1677.84,E2 -1677.84} C_VEL
LIN {X 0,Y 580.746,Z 367.955,A -85,B 0,C 180,E1 -1680.682,E2 -1680.682} C_VEL
LIN {X 0,Y 581.875,Z 373.998,A -85,B 0,C 180,E1 -1680.802,E2 -1680.802} C_VEL
LIN {X 0,Y 581.514,Z 532.884,A -85,B 0,C 180,E1 -1682.831,E2 -1682.831} C_VEL
LIN {X 0,Y 581.439,Z 548.194,A -85,B 0,C 180,E1 -1683.167,E2 -1683.167} C_VEL
LIN {X 0,Y 581.254,Z 563.146,A -85,B 0,C 180,E1 -1683.64,E2 -1683.64} C_VEL
LIN {X 0,Y 581.111,Z 577.401,A -85,B 0,C 180,E1 -1684.238,E2 -1684.238} C_VEL
LIN {X 0,Y 580.919,Z 590.89,A -85,B 0,C 180,E1 -1684.948,E2 -1684.948} C_VEL
LIN {X 0,Y 580.783,Z 604.09,A -85,B 0,C 180,E1 -1685.8,E2 -1685.8} C_VEL
LIN {X 0,Y 580.634,Z 616.154,A -85,B 0,C 180,E1 -1686.738,E2 -1686.738} C_VEL
LIN {X 0,Y 580.484,Z 627.306,A -85,B 0,C 180,E1 -1687.769,E2 -1687.769} C_VEL
LIN {X 0,Y 580.337,Z 637.739,A -85,B 0,C 180,E1 -1688.914,E2 -1688.914} C_VEL
LIN {X 0,Y 580.248,Z 647.344,A -85,B 0,C 180,E1 -1690.176,E2 -1690.176} C_VEL
LIN {X 0,Y 580.182,Z 655.441,A -85,B 0,C 180,E1 -1691.459,E2 -1691.459} C_VEL
LIN {X 0,Y 580.142,Z 662.075,A -85,B 0,C 180,E1 -1692.735,E2 -1692.735} C_VEL
LIN {X 0,Y 580.093,Z 668.092,A -85,B 0,C 180,E1 -1694.181,E2 -1694.181} C_VEL
LIN {X 0,Y 580.07,Z 671.629,A -85,B 0,C 180,E1 -1695.26,E2 -1695.26} C_VEL
LIN {X 0,Y 580.065,Z 675.132,A -85,B 0,C 180,E1 -1696.691,E2 -1696.691} C_VEL
LIN {X 0,Y 580.054,Z 677.364,A -85,B 0,C 180,E1 -1698.113,E2 -1698.113} C_VEL
LIN {X 0,Y 580.058,Z 678.39,A -85,B 0,C 180,E1 -1699.529,E2 -1699.529} C_VEL
LIN {X 0,Y 580.022,Z 678.247,A -85,B 0,C 180,E1 -1700.937,E2 -1700.937} C_VEL
LIN {X 0,Y 580.053,Z 676.944,A -85,B 0,C 180,E1 -1702.341,E2 -1702.341} C_VEL
LIN {X 0,Y 580.065,Z 674.428,A -85,B 0,C 180,E1 -1703.74,E2 -1703.74} C_VEL
LIN {X 0,Y 580.043,Z 670.703,A -85,B 0,C 180,E1 -1705.135,E2 -1705.135} C_VEL
LIN {X 0,Y 580.126,Z 665.699,A -85,B 0,C 180,E1 -1706.527,E2 -1706.527} C_VEL
LIN {X 0,Y 580.124,Z 659.319,A -85,B 0,C 180,E1 -1707.917,E2 -1707.917} C_VEL
LIN {X 0,Y 580.228,Z 651.372,A -85,B 0,C 180,E1 -1709.306,E2 -1709.306} C_VEL
LIN {X 0,Y 580.288,Z 642.954,A -85,B 0,C 180,E1 -1710.52,E2 -1710.52} C_VEL
LIN {X 0,Y 580.45,Z 632.871,A -85,B 0,C 180,E1 -1711.735,E2 -1711.735} C_VEL
LIN {X 0,Y 580.536,Z 622.641,A -85,B 0,C 180,E1 -1712.776,E2 -1712.776} C_VEL
LIN {X 0,Y 580.701,Z 610.445,A -85,B 0,C 180,E1 -1713.817,E2 -1713.817} C_VEL
LIN {X 0,Y 580.896,Z 598.289,A -85,B 0,C 180,E1 -1714.684,E2 -1714.684} C_VEL
LIN {X 0,Y 581.009,Z 585.107,A -85,B 0,C 180,E1 -1715.466,E2 -1715.466} C_VEL
LIN {X 0,Y 581.202,Z 570.478,A -85,B 0,C 180,E1 -1716.161,E2 -1716.161} C_VEL
LIN {X 0,Y 581.345,Z 556.394,A -85,B 0,C 180,E1 -1716.682,E2 -1716.682} C_VEL
LIN {X 0,Y 581.484,Z 541.176,A -85,B 0,C 180,E1 -1717.095,E2 -1717.095} C_VEL
LIN {X 0,Y 581.516,Z 526.898,A -85,B 0,C 180,E1 -1717.349,E2 -1717.349} C_VEL
LIN {X 0,Y 581.879,Z 373.322,A -85,B 0,C 180,E1 -1719.297,E2 -1719.297} C_VEL
LIN {X 0,Y 580.726,Z 367.833,A -85,B 0,C 180,E1 -1719.425,E2 -1719.425} C_VEL
LIN {X 0,Y 581.004,Z 347.504,A -85,B 0,C 180,E1 -1722.221,E2 -1722.221} C_VEL
LIN {X 0,Y 580.376,Z 342.506,A -85,B 0,C 180,E1 -1722.946,E2 -1722.946} C_VEL
LIN {X 0,Y 580.257,Z 341.834,A -85,B 0,C 180,E1 -1723.082,E2 -1723.082} C_VEL
LIN {X 0,Y 580.279,Z 341.832,A -85,B 0,C 180,E1 -1725.453,E2 -1725.453} C_VEL
LIN {X 0,Y 580.249,Z 341.827,A -85,B 0,C 180,E1 -1728.356,E2 -1728.356} C_VEL
LIN {X 0,Y 580.307,Z 341.823,A -85,B 0,C 180,E1 -1731.165,E2 -1731.165} C_VEL
LIN {X 0,Y 580.263,Z 341.834,A -85,B 0,C 180,E1 -1733.559,E2 -1733.559} C_VEL
LIN {X 0,Y 580.267,Z 341.824,A -85,B 0,C 180,E1 -1736.328,E2 -1736.328} C_VEL
LIN {X 0,Y 580.281,Z 341.828,A -85,B 0,C 180,E1 -1739.305,E2 -1739.305} C_VEL
LIN {X 0,Y 580.298,Z 341.82,A -85,B 0,C 180,E1 -1742.201,E2 -1742.201} C_VEL
LIN {X 0,Y 580.282,Z 341.822,A -85,B 0,C 180,E1 -1744.697,E2 -1744.697} C_VEL
LIN {X 0,Y 580.277,Z 341.827,A -85,B 0,C 180,E1 -1747.27,E2 -1747.27} C_VEL
LIN {X 0,Y 580.288,Z 341.82,A -85,B 0,C 180,E1 -1750.269,E2 -1750.269} C_VEL
LIN {X 0,Y 580.256,Z 341.825,A -85,B 0,C 180,E1 -1752.709,E2 -1752.709} C_VEL
LIN {X 0,Y 580.254,Z 341.833,A -85,B 0,C 180,E1 -1755.611,E2 -1755.611} C_VEL
LIN {X 0,Y 580.254,Z 341.826,A -85,B 0,C 180,E1 -1758.228,E2 -1758.228} C_VEL
LIN {X 0,Y 580.268,Z 341.825,A -85,B 0,C 180,E1 -1760.964,E2 -1760.964} C_VEL
LIN {X 0,Y 580.245,Z 341.836,A -85,B 0,C 180,E1 -1763.594,E2 -1763.594} C_VEL
LIN {X 0,Y 580.31,Z 341.82,A -85,B 0,C 180,E1 -1766.144,E2 -1766.144} C_VEL
LIN {X 0,Y 580.272,Z 341.823,A -85,B 0,C 180,E1 -1768.614,E2 -1768.614} C_VEL
LIN {X 0,Y 580.29,Z 341.822,A -85,B 0,C 180,E1 -1771.023,E2 -1771.023} C_VEL
LIN {X 0,Y 580.252,Z 341.823,A -85,B 0,C 180,E1 -1774.149,E2 -1774.149} C_VEL
LIN {X 0,Y 580.272,Z 341.821,A -85,B 0,C 180,E1 -1776.441,E2 -1776.441} C_VEL
LIN {X 0,Y 580.272,Z 341.831,A -85,B 0,C 180,E1 -1779.437,E2 -1779.437} C_VEL
LIN {X 0,Y 580.256,Z 341.833,A -85,B 0,C 180,E1 -1781.644,E2 -1781.644} C_VEL
LIN {X 0,Y 580.261,Z 341.83,A -85,B 0,C 180,E1 -1783.825,E2 -1783.825} C_VEL
LIN {X 0,Y 580.314,Z 341.821,A -85,B 0,C 180,E1 -1785.982,E2 -1785.982} C_VEL
LIN {X 0,Y 580.31,Z 341.817,A -85,B 0,C 180,E1 -1788.827,E2 -1788.827} C_VEL
LIN {X 0,Y 580.309,Z 341.828,A -85,B 0,C 180,E1 -1791.643,E2 -1791.643} C_VEL
LIN {X 0,Y 580.303,Z 341.817,A -85,B 0,C 180,E1 -1794.44,E2 -1794.44} C_VEL
LIN {X 0,Y 580.323,Z 341.82,A -85,B 0,C 180,E1 -1797.223,E2 -1797.223} C_VEL
LIN {X 0,Y 580.352,Z 341.816,A -85,B 0,C 180,E1 -1800,E2 -1800} C_VEL
LIN {X 0,Y 580.317,Z 341.816,A -85,B 0,C 180,E1 -1802.776,E2 -1802.776} C_VEL
LIN {X 0,Y 580.312,Z 341.828,A -85,B 0,C 180,E1 -1805.56,E2 -1805.56} C_VEL
LIN {X 0,Y 580.306,Z 341.818,A -85,B 0,C 180,E1 -1808.356,E2 -1808.356} C_VEL
LIN {X 0,Y 580.304,Z 341.822,A -85,B 0,C 180,E1 -1811.191,E2 -1811.191} C_VEL
LIN {X 0,Y 580.299,Z 341.82,A -85,B 0,C 180,E1 -1814.331,E2 -1814.331} C_VEL
LIN {X 0,Y 580.251,Z 341.826,A -85,B 0,C 180,E1 -1816.899,E2 -1816.899} C_VEL
LIN {X 0,Y 580.278,Z 341.828,A -85,B 0,C 180,E1 -1819.823,E2 -1819.823} C_VEL
LIN {X 0,Y 580.253,Z 341.828,A -85,B 0,C 180,E1 -1822.053,E2 -1822.053} C_VEL
LIN {X 0,Y 580.288,Z 341.823,A -85,B 0,C 180,E1 -1825.08,E2 -1825.08} C_VEL
LIN {X 0,Y 580.248,Z 341.828,A -85,B 0,C 180,E1 -1828.188,E2 -1828.188} C_VEL
LIN {X 0,Y 580.27,Z 341.823,A -85,B 0,C 180,E1 -1830.692,E2 -1830.692} C_VEL
LIN {X 0,Y 580.301,Z 341.824,A -85,B 0,C 180,E1 -1833.315,E2 -1833.315} C_VEL
LIN {X 0,Y 580.231,Z 341.836,A -85,B 0,C 180,E1 -1835.754,E2 -1835.754} C_VEL
LIN {X 0,Y 580.278,Z 341.824,A -85,B 0,C 180,E1 -1838.147,E2 -1838.147} C_VEL
LIN {X 0,Y 580.278,Z 341.822,A -85,B 0,C 180,E1 -1840.845,E2 -1840.845} C_VEL
LIN {X 0,Y 580.236,Z 341.838,A -85,B 0,C 180,E1 -1843.662,E2 -1843.662} C_VEL
LIN {X 0,Y 580.241,Z 341.827,A -85,B 0,C 180,E1 -1846.613,E2 -1846.613} C_VEL
LIN {X 0,Y 580.277,Z 341.826,A -85,B 0,C 180,E1 -1849.155,E2 -1849.155} C_VEL
LIN {X 0,Y 580.28,Z 341.828,A -85,B 0,C 180,E1 -1851.928,E2 -1851.928} C_VEL
LIN {X 0,Y 580.226,Z 341.829,A -85,B 0,C 180,E1 -1854.451,E2 -1854.451} C_VEL
LIN {X 0,Y 580.286,Z 341.823,A -85,B 0,C 180,E1 -1856.975,E2 -1856.975} C_VEL
LIN {X 0,Y 580.29,Z 341.828,A -85,B 0,C 180,E1 -1859.425,E2 -1859.425} C_VEL
LIN {X 0,Y 580.256,Z 341.831,A -85,B 0,C 180,E1 -1862.149,E2 -1862.149} C_VEL
LIN {X 0,Y 580.286,Z 341.964,A -85,B 0,C 180,E1 -1863.773,E2 -1863.773} C_VEL
LIN {X 0,Y 581.36,Z 346.597,A -85,B 0,C 180,E1 -1864.394,E2 -1864.394} C_VEL
LIN {X 0,Y 581.29,Z 362.273,A -85,B 0,C 180,E1 -1866.296,E2 -1866.296} C_VEL
LIN {X 0,Y 581.059,Z 385.789,A -85,B 0,C 180,E1 -1869.096,E2 -1869.096} C_VEL
LIN {X 0,Y 580.898,Z 398.876,A -85,B 0,C 180,E1 -1870.631,E2 -1870.631} C_VEL
LIN {X 0,Y 581.879,Z 404.739,A -85,B 0,C 180,E1 -1870.741,E2 -1870.741} C_VEL
LIN {X 0,Y 581.529,Z 565.478,A -85,B 0,C 180,E1 -1872.797,E2 -1872.797} C_VEL
LIN {X 0,Y 581.412,Z 580.703,A -85,B 0,C 180,E1 -1873.136,E2 -1873.136} C_VEL
LIN {X 0,Y 581.234,Z 596.04,A -85,B 0,C 180,E1 -1873.627,E2 -1873.627} C_VEL
LIN {X 0,Y 581.125,Z 609.765,A -85,B 0,C 180,E1 -1874.21,E2 -1874.21} C_VEL
LIN {X 0,Y 580.943,Z 623.239,A -85,B 0,C 180,E1 -1874.924,E2 -1874.924} C_VEL
LIN {X 0,Y 580.805,Z 636.478,A -85,B 0,C 180,E1 -1875.783,E2 -1875.783} C_VEL
LIN {X 0,Y 580.608,Z 648.287,A -85,B 0,C 180,E1 -1876.704,E2 -1876.704} C_VEL
LIN {X 0,Y 580.479,Z 659.748,A -85,B 0,C 180,E1 -1877.768,E2 -1877.768} C_VEL
LIN {X 0,Y 580.307,Z 670.454,A -85,B 0,C 180,E1 -1878.954,E2 -1878.954} C_VEL
LIN {X 0,Y 580.269,Z 678.856,A -85,B 0,C 180,E1 -1880.061,E2 -1880.061} C_VEL
LIN {X 0,Y 580.213,Z 686.732,A -85,B 0,C 180,E1 -1881.291,E2 -1881.291} C_VEL
LIN {X 0,Y 580.13,Z 694.088,A -85,B 0,C 180,E1 -1882.692,E2 -1882.692} C_VEL
LIN {X 0,Y 580.131,Z 699.923,A -85,B 0,C 180,E1 -1884.09,E2 -1884.09} C_VEL
LIN {X 0,Y 580.041,Z 703.384,A -85,B 0,C 180,E1 -1885.135,E2 -1885.135} C_VEL
LIN {X 0,Y 580.105,Z 706.888,A -85,B 0,C 180,E1 -1886.527,E2 -1886.527} C_VEL
LIN {X 0,Y 580.038,Z 709.193,A -85,B 0,C 180,E1 -1887.917,E2 -1887.917} C_VEL
LIN {X 0,Y 580.036,Z 710.349,A -85,B 0,C 180,E1 -1889.306,E2 -1889.306} C_VEL
LIN {X 0,Y 580.036,Z 710.349,A -85,B 0,C 180,E1 -1890.694,E2 -1890.694} C_VEL
LIN {X 0,Y 580.038,Z 709.192,A -85,B 0,C 180,E1 -1892.083,E2 -1892.083} C_VEL
LIN {X 0,Y 580.105,Z 706.887,A -85,B 0,C 180,E1 -1893.473,E2 -1893.473} C_VEL
LIN {X 0,Y 580.041,Z 703.385,A -85,B 0,C 180,E1 -1894.865,E2 -1894.865} C_VEL
LIN {X 0,Y 580.092,Z 698.608,A -85,B 0,C 180,E1 -1896.26,E2 -1896.26} C_VEL
LIN {X 0,Y 580.165,Z 692.424,A -85,B 0,C 180,E1 -1897.658,E2 -1897.658} C_VEL
LIN {X 0,Y 580.207,Z 684.65,A -85,B 0,C 180,E1 -1899.06,E2 -1899.06} C_VEL
LIN {X 0,Y 580.309,Z 676.369,A -85,B 0,C 180,E1 -1900.29,E2 -1900.29} C_VEL
LIN {X 0,Y 580.382,Z 666.395,A -85,B 0,C 180,E1 -1901.525,E2 -1901.525} C_VEL
LIN {X 0,Y 580.541,Z 656.19,A -85,B 0,C 180,E1 -1902.586,E2 -1902.586} C_VEL
LIN {X 0,Y 580.678,Z 644.018,A -85,B 0,C 180,E1 -1903.651,E2 -1903.651} C_VEL
LIN {X 0,Y 580.846,Z 631.804,A -85,B 0,C 180,E1 -1904.542,E2 -1904.542} C_VEL
LIN {X 0,Y 580.972,Z 618.518,A -85,B 0,C 180,E1 -1905.344,E2 -1905.344} C_VEL
LIN {X 0,Y 581.199,Z 603.834,A -85,B 0,C 180,E1 -1906.058,E2 -1906.058} C_VEL
LIN {X 0,Y 581.337,Z 589.615,A -85,B 0,C 180,E1 -1906.595,E2 -1906.595} C_VEL
LIN {X 0,Y 581.475,Z 574.588,A -85,B 0,C 180,E1 -1907.015,E2 -1907.015} C_VEL
LIN {X 0,Y 581.529,Z 559.397,A -85,B 0,C 180,E1 -1907.296,E2 -1907.296} C_VEL
LIN {X 0,Y 581.802,Z 403.624,A -85,B 0,C 180,E1 -1909.276,E2 -1909.276} C_VEL
LIN {X 0,Y 580.922,Z 398.728,A -85,B 0,C 180,E1 -1909.386,E2 -1909.386} C_VEL
LIN {X 0,Y 581.199,Z 373.248,A -85,B 0,C 180,E1 -1912.39,E2 -1912.39} C_VEL
LIN {X 0,Y 581.455,Z 349.733,A -85,B 0,C 180,E1 -1915.218,E2 -1915.218} C_VEL
LIN {X 0,Y 581.358,Z 346.597,A -85,B 0,C 180,E1 -1915.606,E2 -1915.606} C_VEL
LIN {X 0,Y 580.273,Z 341.833,A -85,B 0,C 180,E1 -1916.255,E2 -1916.255} C_VEL
LIN {X 0,Y 580.278,Z 341.823,A -85,B 0,C 180,E1 -1919.306,E2 -1919.306} C_VEL
LIN {X 0,Y 580.295,Z 341.829,A -85,B 0,C 180,E1 -1922.201,E2 -1922.201} C_VEL
LIN {X 0,Y 580.275,Z 341.828,A -85,B 0,C 180,E1 -1924.697,E2 -1924.697} C_VEL
LIN {X 0,Y 580.271,Z 341.823,A -85,B 0,C 180,E1 -1927.271,E2 -1927.271} C_VEL
LIN {X 0,Y 580.284,Z 341.83,A -85,B 0,C 180,E1 -1930.27,E2 -1930.27} C_VEL
LIN {X 0,Y 580.269,Z 341.828,A -85,B 0,C 180,E1 -1932.707,E2 -1932.707} C_VEL
LIN {X 0,Y 580.25,Z 341.826,A -85,B 0,C 180,E1 -1935.611,E2 -1935.611} C_VEL
LIN {X 0,Y 580.249,Z 341.834,A -85,B 0,C 180,E1 -1938.229,E2 -1938.229} C_VEL
LIN {X 0,Y 580.266,Z 341.826,A -85,B 0,C 180,E1 -1940.964,E2 -1940.964} C_VEL
LIN {X 0,Y 580.24,Z 341.825,A -85,B 0,C 180,E1 -1943.595,E2 -1943.595} C_VEL
LIN {X 0,Y 580.309,Z 341.824,A -85,B 0,C 180,E1 -1946.145,E2 -1946.145} C_VEL
LIN {X 0,Y 580.266,Z 341.827,A -85,B 0,C 180,E1 -1948.614,E2 -1948.614} C_VEL
LIN {X 0,Y 580.283,Z 341.823,A -85,B 0,C 180,E1 -1951.024,E2 -1951.024} C_VEL
LIN {X 0,Y 580.266,Z 341.829,A -85,B 0,C 180,E1 -1954.15,E2 -1954.15} C_VEL
LIN {X 0,Y 580.258,Z 341.826,A -85,B 0,C 180,E1 -1957,E2 -1957} C_VEL
LIN {X 0,Y 580.264,Z 341.824,A -85,B 0,C 180,E1 -1959.437,E2 -1959.437} C_VEL
LIN {X 0,Y 580.246,Z 341.826,A -85,B 0,C 180,E1 -1961.645,E2 -1961.645} C_VEL
LIN {X 0,Y 580.276,Z 341.831,A -85,B 0,C 180,E1 -1964.547,E2 -1964.547} C_VEL
LIN {X 0,Y 580.25,Z 341.831,A -85,B 0,C 180,E1 -1966.696,E2 -1966.696} C_VEL
LIN {X 0,Y 580.308,Z 341.822,A -85,B 0,C 180,E1 -1968.827,E2 -1968.827} C_VEL
LIN {X 0,Y 580.307,Z 341.818,A -85,B 0,C 180,E1 -1971.644,E2 -1971.644} C_VEL
LIN {X 0,Y 580.314,Z 341.828,A -85,B 0,C 180,E1 -1974.44,E2 -1974.44} C_VEL
LIN {X 0,Y 580.319,Z 341.818,A -85,B 0,C 180,E1 -1977.224,E2 -1977.224} C_VEL
LIN {X 0,Y 580.352,Z 341.815,A -85,B 0,C 180,E1 -1980,E2 -1980} C_VEL
LIN {X 0,Y 580.328,Z 341.82,A -85,B 0,C 180,E1 -1982.777,E2 -1982.777} C_VEL
LIN {X 0,Y 580.306,Z 341.819,A -85,B 0,C 180,E1 -1985.56,E2 -1985.56} C_VEL
LIN {X 0,Y 580.31,Z 341.826,A -85,B 0,C 180,E1 -1988.357,E2 -1988.357} C_VEL
LIN {X 0,Y 580.304,Z 341.819,A -85,B 0,C 180,E1 -1991.191,E2 -1991.191} C_VEL
LIN {X 0,Y 580.324,Z 341.819,A -85,B 0,C 180,E1 -1994.017,E2 -1994.017} C_VEL
LIN {X 0,Y 580.317,Z 341.821,A -85,B 0,C 180,E1 -1996.914,E2 -1996.914} C_VEL
LIN {X 0,Y 580.285,Z 341.819,A -85,B 0,C 180,E1 -1999.823,E2 -1999.823} C_VEL
LIN {X 0,Y 580.285,Z 341.821,A -85,B 0,C 180,E1 -2001.328,E2 -2001.328} C_VEL
LIN {X 0,Y 579.586,Z 341.91,A -85,B 0,C 180,E1 -2001.907,E2 -2001.907} C_VEL
LIN {X 0,Y 576.711,Z 342.271,A -85,B 0,C 180,E1 -2002.847,E2 -2002.847} C_VEL
LIN {X 0,Y 574.312,Z 342.567,A -85,B 0,C 180,E1 -2003.603,E2 -2003.603} C_VEL
LIN {X 0,Y 573.301,Z 342.696,A -85,B 0,C 180,E1 -2004.187,E2 -2004.187} C_VEL
LIN {X 0,Y 573.228,Z 342.703,A -85,B 0,C 180,E1 -2004.384,E2 -2004.384} C_VEL
LIN {X 0,Y 573.191,Z 342.708,A -85,B 0,C 180,E1 -2006.979,E2 -2006.979} C_VEL
LIN {X 0,Y 573.245,Z 342.698,A -85,B 0,C 180,E1 -2009.487,E2 -2009.487} C_VEL
LIN {X 0,Y 573.255,Z 342.706,A -85,B 0,C 180,E1 -2012.645,E2 -2012.645} C_VEL
LIN {X 0,Y 573.196,Z 342.703,A -85,B 0,C 180,E1 -2015.189,E2 -2015.189} C_VEL
LIN {X 0,Y 573.225,Z 342.702,A -85,B 0,C 180,E1 -2017.809,E2 -2017.809} C_VEL
LIN {X 0,Y 573.249,Z 342.707,A -85,B 0,C 180,E1 -2020.525,E2 -2020.525} C_VEL
LIN {X 0,Y 573.211,Z 342.703,A -85,B 0,C 180,E1 -2023.362,E2 -2023.362} C_VEL
LIN {X 0,Y 573.239,Z 342.706,A -85,B 0,C 180,E1 -2026.332,E2 -2026.332} C_VEL
LIN {X 0,Y 573.249,Z 342.699,A -85,B 0,C 180,E1 -2029.475,E2 -2029.475} C_VEL
LIN {X 0,Y 573.233,Z 342.705,A -85,B 0,C 180,E1 -2032.192,E2 -2032.192} C_VEL
LIN {X 0,Y 573.231,Z 342.704,A -85,B 0,C 180,E1 -2035.23,E2 -2035.23} C_VEL
LIN {X 0,Y 573.281,Z 342.799,A -85,B 0,C 180,E1 -2036.886,E2 -2036.886} C_VEL
LIN {X 0,Y 574.038,Z 347.954,A -85,B 0,C 180,E1 -2037.649,E2 -2037.649} C_VEL
LIN {X 0,Y 573.832,Z 367.885,A -85,B 0,C 180,E1 -2040.43,E2 -2040.43} C_VEL
LIN {X 0,Y 575.176,Z 375.266,A -85,B 0,C 180,E1 -2040.585,E2 -2040.585} C_VEL
LIN {X 0,Y 574.737,Z 532.754,A -85,B 0,C 180,E1 -2042.62,E2 -2042.62} C_VEL
LIN {X 0,Y 574.639,Z 548.102,A -85,B 0,C 180,E1 -2042.959,E2 -2042.959} C_VEL
LIN {X 0,Y 574.438,Z 563.151,A -85,B 0,C 180,E1 -2043.44,E2 -2043.44} C_VEL
LIN {X 0,Y 574.25,Z 577.605,A -85,B 0,C 180,E1 -2044.054,E2 -2044.054} C_VEL
LIN {X 0,Y 574.038,Z 590.486,A -85,B 0,C 180,E1 -2044.74,E2 -2044.74} C_VEL
LIN {X 0,Y 573.845,Z 603.537,A -85,B 0,C 180,E1 -2045.585,E2 -2045.585} C_VEL
LIN {X 0,Y 573.677,Z 616.419,A -85,B 0,C 180,E1 -2046.596,E2 -2046.596} C_VEL
LIN {X 0,Y 573.466,Z 627.856,A -85,B 0,C 180,E1 -2047.672,E2 -2047.672} C_VEL
LIN {X 0,Y 573.291,Z 637.121,A -85,B 0,C 180,E1 -2048.701,E2 -2048.701} C_VEL
LIN {X 0,Y 573.229,Z 646.436,A -85,B 0,C 180,E1 -2049.923,E2 -2049.923} C_VEL
LIN {X 0,Y 573.117,Z 653.936,A -85,B 0,C 180,E1 -2051.088,E2 -2051.088} C_VEL
LIN {X 0,Y 573.073,Z 661.486,A -85,B 0,C 180,E1 -2052.515,E2 -2052.515} C_VEL
LIN {X 0,Y 573.031,Z 667.644,A -85,B 0,C 180,E1 -2053.981,E2 -2053.981} C_VEL
LIN {X 0,Y 572.98,Z 671.247,A -85,B 0,C 180,E1 -2055.073,E2 -2055.073} C_VEL
LIN {X 0,Y 572.976,Z 674.875,A -85,B 0,C 180,E1 -2056.523,E2 -2056.523} C_VEL
LIN {X 0,Y 572.948,Z 677.222,A -85,B 0,C 180,E1 -2057.964,E2 -2057.964} C_VEL
LIN {X 0,Y 572.984,Z 678.362,A -85,B 0,C 180,E1 -2059.398,E2 -2059.398} C_VEL
LIN {X 0,Y 572.922,Z 678.325,A -85,B 0,C 180,E1 -2060.824,E2 -2060.824} C_VEL
LIN {X 0,Y 572.968,Z 677.088,A -85,B 0,C 180,E1 -2062.246,E2 -2062.246} C_VEL
LIN {X 0,Y 572.973,Z 674.682,A -85,B 0,C 180,E1 -2063.662,E2 -2063.662} C_VEL
LIN {X 0,Y 572.952,Z 671.074,A -85,B 0,C 180,E1 -2065.074,E2 -2065.074} C_VEL
LIN {X 0,Y 573.057,Z 666.194,A -85,B 0,C 180,E1 -2066.484,E2 -2066.484} C_VEL
LIN {X 0,Y 573.038,Z 659.95,A -85,B 0,C 180,E1 -2067.891,E2 -2067.891} C_VEL
LIN {X 0,Y 573.159,Z 652.148,A -85,B 0,C 180,E1 -2069.297,E2 -2069.297} C_VEL
LIN {X 0,Y 573.24,Z 643.892,A -85,B 0,C 180,E1 -2070.527,E2 -2070.527} C_VEL
LIN {X 0,Y 573.411,Z 633.998,A -85,B 0,C 180,E1 -2071.756,E2 -2071.756} C_VEL
LIN {X 0,Y 573.552,Z 623.962,A -85,B 0,C 180,E1 -2072.809,E2 -2072.809} C_VEL
LIN {X 0,Y 573.733,Z 612.033,A -85,B 0,C 180,E1 -2073.863,E2 -2073.863} C_VEL
LIN {X 0,Y 573.98,Z 598.848,A -85,B 0,C 180,E1 -2074.829,E2 -2074.829} C_VEL
LIN {X 0,Y 574.12,Z 585.771,A -85,B 0,C 180,E1 -2075.62,E2 -2075.62} C_VEL
LIN {X 0,Y 574.343,Z 571.328,A -85,B 0,C 180,E1 -2076.323,E2 -2076.323} C_VEL
LIN {X 0,Y 574.521,Z 557.409,A -85,B 0,C 180,E1 -2076.85,E2 -2076.85} C_VEL
LIN {X 0,Y 574.658,Z 542.896,A -85,B 0,C 180,E1 -2077.26,E2 -2077.26} C_VEL
LIN {X 0,Y 574.75,Z 528.935,A -85,B 0,C 180,E1 -2077.528,E2 -2077.528} C_VEL
LIN {X 0,Y 575.167,Z 374.298,A -85,B 0,C 180,E1 -2079.518,E2 -2079.518} C_VEL
LIN {X 0,Y 573.774,Z 367.962,A -85,B 0,C 180,E1 -2079.652,E2 -2079.652} C_VEL
LIN {X 0,Y 574.099,Z 348.438,A -85,B 0,C 180,E1 -2082.371,E2 -2082.371} C_VEL
LIN {X 0,Y 573.236,Z 342.71,A -85,B 0,C 180,E1 -2083.245,E2 -2083.245} C_VEL
LIN {X 0,Y 573.218,Z 342.711,A -85,B 0,C 180,E1 -2085.648,E2 -2085.648} C_VEL
LIN {X 0,Y 573.224,Z 342.707,A -85,B 0,C 180,E1 -2087.849,E2 -2087.849} C_VEL
LIN {X 0,Y 573.239,Z 342.701,A -85,B 0,C 180,E1 -2090.077,E2 -2090.077} C_VEL
LIN {X 0,Y 573.225,Z 342.702,A -85,B 0,C 180,E1 -2092.338,E2 -2092.338} C_VEL
LIN {X 0,Y 573.238,Z 342.708,A -85,B 0,C 180,E1 -2095.411,E2 -2095.411} C_VEL
LIN {X 0,Y 573.211,Z 342.703,A -85,B 0,C 180,E1 -2098.566,E2 -2098.566} C_VEL
LIN {X 0,Y 573.222,Z 342.703,A -85,B 0,C 180,E1 -2100.994,E2 -2100.994} C_VEL
LIN {X 0,Y 573.269,Z 342.704,A -85,B 0,C 180,E1 -2103.524,E2 -2103.524} C_VEL
LIN {X 0,Y 573.192,Z 342.706,A -85,B 0,C 180,E1 -2106.053,E2 -2106.053} C_VEL
LIN {X 0,Y 573.237,Z 342.7,A -85,B 0,C 180,E1 -2108.702,E2 -2108.702} C_VEL
LIN {X 0,Y 573.21,Z 342.71,A -85,B 0,C 180,E1 -2111.459,E2 -2111.459} C_VEL
LIN {X 0,Y 573.221,Z 342.701,A -85,B 0,C 180,E1 -2114.335,E2 -2114.335} C_VEL
LIN {X 0,Y 573.234,Z 342.705,A -85,B 0,C 180,E1 -2117.359,E2 -2117.359} C_VEL
LIN {X 0,Y 573.236,Z 342.699,A -85,B 0,C 180,E1 -2120.391,E2 -2120.391} C_VEL
LIN {X 0,Y 573.225,Z 342.703,A -85,B 0,C 180,E1 -2123.075,E2 -2123.075} C_VEL
LIN {X 0,Y 573.262,Z 342.704,A -85,B 0,C 180,E1 -2125.67,E2 -2125.67} C_VEL
LIN {X 0,Y 573.24,Z 342.701,A -85,B 0,C 180,E1 -2128.184,E2 -2128.184} C_VEL
LIN {X 0,Y 573.244,Z 342.697,A -85,B 0,C 180,E1 -2130.633,E2 -2130.633} C_VEL
LIN {X 0,Y 573.203,Z 342.707,A -85,B 0,C 180,E1 -2133.515,E2 -2133.515} C_VEL
LIN {X 0,Y 573.223,Z 342.701,A -85,B 0,C 180,E1 -2136.134,E2 -2136.134} C_VEL
LIN {X 0,Y 573.252,Z 342.701,A -85,B 0,C 180,E1 -2139.173,E2 -2139.173} C_VEL
LIN {X 0,Y 573.212,Z 342.709,A -85,B 0,C 180,E1 -2141.41,E2 -2141.41} C_VEL
LIN {X 0,Y 573.239,Z 342.709,A -85,B 0,C 180,E1 -2143.621,E2 -2143.621} C_VEL
LIN {X 0,Y 573.26,Z 342.702,A -85,B 0,C 180,E1 -2145.806,E2 -2145.806} C_VEL
LIN {X 0,Y 573.267,Z 342.693,A -85,B 0,C 180,E1 -2148.745,E2 -2148.745} C_VEL
LIN {X 0,Y 573.252,Z 342.706,A -85,B 0,C 180,E1 -2151.54,E2 -2151.54} C_VEL
LIN {X 0,Y 573.272,Z 342.693,A -85,B 0,C 180,E1 -2154.371,E2 -2154.371} C_VEL
LIN {X 0,Y 573.312,Z 342.695,A -85,B 0,C 180,E1 -2157.892,E2 -2157.892} C_VEL
LIN {X 0,Y 573.321,Z 342.691,A -85,B 0,C 180,E1 -2160,E2 -2160} C_VEL
LIN {X 0,Y 573.286,Z 342.692,A -85,B 0,C 180,E1 -2162.81,E2 -2162.81} C_VEL
LIN {X 0,Y 573.279,Z 342.704,A -85,B 0,C 180,E1 -2165.628,E2 -2165.628} C_VEL
LIN {X 0,Y 573.249,Z 342.697,A -85,B 0,C 180,E1 -2168.46,E2 -2168.46} C_VEL
LIN {X 0,Y 573.275,Z 342.7,A -85,B 0,C 180,E1 -2171.312,E2 -2171.312} C_VEL
LIN {X 0,Y 573.273,Z 342.694,A -85,B 0,C 180,E1 -2174.42,E2 -2174.42} C_VEL
LIN {X 0,Y 573.196,Z 342.706,A -85,B 0,C 180,E1 -2177.113,E2 -2177.113} C_VEL
LIN {X 0,Y 573.234,Z 342.702,A -85,B 0,C 180,E1 -2180.077,E2 -2180.077} C_VEL
LIN {X 0,Y 573.22,Z 342.701,A -85,B 0,C 180,E1 -2182.338,E2 -2182.338} C_VEL
LIN {X 0,Y 573.235,Z 342.706,A -85,B 0,C 180,E1 -2185.411,E2 -2185.411} C_VEL
LIN {X 0,Y 573.206,Z 342.703,A -85,B 0,C 180,E1 -2188.566,E2 -2188.566} C_VEL
LIN {X 0,Y 573.218,Z 342.703,A -85,B 0,C 180,E1 -2190.994,E2 -2190.994} C_VEL
LIN {X 0,Y 573.264,Z 342.704,A -85,B 0,C 180,E1 -2193.524,E2 -2193.524} C_VEL
LIN {X 0,Y 573.187,Z 342.709,A -85,B 0,C 180,E1 -2196.053,E2 -2196.053} C_VEL
LIN {X 0,Y 573.233,Z 342.699,A -85,B 0,C 180,E1 -2198.702,E2 -2198.702} C_VEL
LIN {X 0,Y 573.204,Z 342.71,A -85,B 0,C 180,E1 -2201.459,E2 -2201.459} C_VEL
LIN {X 0,Y 573.217,Z 342.703,A -85,B 0,C 180,E1 -2204.335,E2 -2204.335} C_VEL
LIN {X 0,Y 573.235,Z 342.706,A -85,B 0,C 180,E1 -2207.359,E2 -2207.359} C_VEL
LIN {X 0,Y 573.232,Z 342.701,A -85,B 0,C 180,E1 -2210.391,E2 -2210.391} C_VEL
LIN {X 0,Y 573.22,Z 342.704,A -85,B 0,C 180,E1 -2213.075,E2 -2213.075} C_VEL
LIN {X 0,Y 573.257,Z 342.707,A -85,B 0,C 180,E1 -2215.67,E2 -2215.67} C_VEL
LIN {X 0,Y 573.236,Z 342.702,A -85,B 0,C 180,E1 -2218.184,E2 -2218.184} C_VEL
LIN {X 0,Y 573.243,Z 342.7,A -85,B 0,C 180,E1 -2220.633,E2 -2220.633} C_VEL
LIN {X 0,Y 573.23,Z 342.84,A -85,B 0,C 180,E1 -2223.548,E2 -2223.548} C_VEL
LIN {X 0,Y 574.639,Z 349.732,A -85,B 0,C 180,E1 -2224.461,E2 -2224.461} C_VEL
LIN {X 0,Y 574.39,Z 370.112,A -85,B 0,C 180,E1 -2226.95,E2 -2226.95} C_VEL
LIN {X 0,Y 574.051,Z 395.195,A -85,B 0,C 180,E1 -2229.952,E2 -2229.952} C_VEL
LIN {X 0,Y 574.016,Z 398.84,A -85,B 0,C 180,E1 -2230.385,E2 -2230.385} C_VEL
LIN {X 0,Y 575.164,Z 404.913,A -85,B 0,C 180,E1 -2230.509,E2 -2230.509} C_VEL
LIN {X 0,Y 574.763,Z 565.006,A -85,B 0,C 180,E1 -2232.58,E2 -2232.58} C_VEL
LIN {X 0,Y 574.626,Z 580.702,A -85,B 0,C 180,E1 -2232.93,E2 -2232.93} C_VEL
LIN {X 0,Y 574.431,Z 596.038,A -85,B 0,C 180,E1 -2233.428,E2 -2233.428} C_VEL
LIN {X 0,Y 574.293,Z 609.768,A -85,B 0,C 180,E1 -2234.017,E2 -2234.017} C_VEL
LIN {X 0,Y 574.048,Z 623.242,A -85,B 0,C 180,E1 -2234.739,E2 -2234.739} C_VEL
LIN {X 0,Y 573.861,Z 636.815,A -85,B 0,C 180,E1 -2235.631,E2 -2235.631} C_VEL
LIN {X 0,Y 573.635,Z 649.348,A -85,B 0,C 180,E1 -2236.629,E2 -2236.629} C_VEL
LIN {X 0,Y 573.478,Z 659.748,A -85,B 0,C 180,E1 -2237.616,E2 -2237.616} C_VEL
LIN {X 0,Y 573.286,Z 669.769,A -85,B 0,C 180,E1 -2238.734,E2 -2238.734} C_VEL
LIN {X 0,Y 573.243,Z 678.857,A -85,B 0,C 180,E1 -2239.938,E2 -2239.938} C_VEL
LIN {X 0,Y 573.132,Z 686.733,A -85,B 0,C 180,E1 -2241.183,E2 -2241.183} C_VEL
LIN {X 0,Y 573.074,Z 694.089,A -85,B 0,C 180,E1 -2242.601,E2 -2242.601} C_VEL
LIN {X 0,Y 573.041,Z 699.923,A -85,B 0,C 180,E1 -2244.016,E2 -2244.016} C_VEL
LIN {X 0,Y 572.951,Z 703.385,A -85,B 0,C 180,E1 -2245.074,E2 -2245.074} C_VEL
LIN {X 0,Y 573.005,Z 706.889,A -85,B 0,C 180,E1 -2246.484,E2 -2246.484} C_VEL
LIN {X 0,Y 572.938,Z 709.192,A -85,B 0,C 180,E1 -2247.891,E2 -2247.891} C_VEL
LIN {X 0,Y 572.936,Z 710.349,A -85,B 0,C 180,E1 -2249.297,E2 -2249.297} C_VEL
LIN {X 0,Y 572.936,Z 710.349,A -85,B 0,C 180,E1 -2250.703,E2 -2250.703} C_VEL
LIN {X 0,Y 572.938,Z 709.191,A -85,B 0,C 180,E1 -2252.109,E2 -2252.109} C_VEL
LIN {X 0,Y 573.005,Z 706.887,A -85,B 0,C 180,E1 -2253.516,E2 -2253.516} C_VEL
LIN {X 0,Y 572.951,Z 703.385,A -85,B 0,C 180,E1 -2254.926,E2 -2254.926} C_VEL
LIN {X 0,Y 573.013,Z 698.608,A -85,B 0,C 180,E1 -2256.337,E2 -2256.337} C_VEL
LIN {X 0,Y 573.094,Z 692.423,A -85,B 0,C 180,E1 -2257.753,E2 -2257.753} C_VEL
LIN {X 0,Y 573.135,Z 684.649,A -85,B 0,C 180,E1 -2259.173,E2 -2259.173} C_VEL
LIN {X 0,Y 573.27,Z 676.369,A -85,B 0,C 180,E1 -2260.418,E2 -2260.418} C_VEL
LIN {X 0,Y 573.385,Z 666.391,A -85,B 0,C 180,E1 -2261.668,E2 -2261.668} C_VEL
